KUKA KRL program: EPS_2_25618_SANMH08_A_20250918115514.src

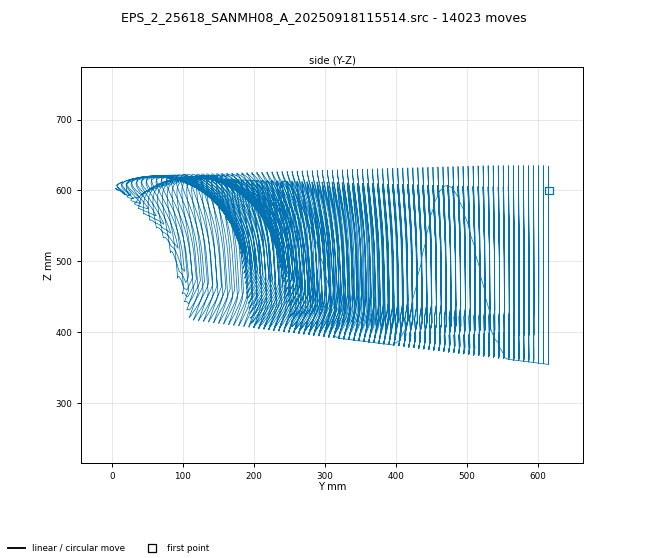
[picture p0: tool path of EPS_2_25618_SANMH08_A_20250918115514.src, 14023 of 14025 moves have a stored position in this frame; points joined in program order, loops and branches not executed]
&ACCESS RVP
&REL 4
&COMMENT QRS 19112012
&PARAM EDITMASK = *
DEF PART()
EXT BAS (BAS_COMMAND :IN,REAL :IN )
INT I
BAS (#INITMOV,0 )

;KUKA QRS Post kuka4.cps  Date:22-06-2017 !

File_ID=2843

QRS_PRE_INIT()

;Init var - Until changes are made in qrs_pre_init
Outlet_Square_prg=0
Inlet_1_Square_prg=0
Inlet_2_Square_prg=0
Inlet_3_Square_prg=0
Inlet_4_Square_prg=0
Inlet_5_Square_prg=0

Outlet_1={X 0.000, Y 530.070, Z 534.500, B 0.000, E1 0.000 }
Inlet_1={X 0.000, Y 532.210, Z 504.500, B 0.000, E1 142.000 }
Inlet_2={X 0.000, Y 532.210, Z 504.500, B 0.000, E1 248.000 }
Outlet_1_type=201
Inlet_1_type=201
Inlet_2_type=201
;QRS#1=Sidecore dimensions
;QRS#2=200-8" PVC SDR 35
;QRS#3=200-8" PVC SDR 35
;QRS#4=200-8" PVC SDR 35
;QRS#5=
;QRS#6=
;QRS#7=
;QRS#8=
;QRS#9=12-08 PSX
;QRS#10=12-08 PSX
;QRS#11=12-08 PSX
;QRS#12=
;QRS#13=
;QRS#14=
;QRS#15=
;QRS#16=1220x127x914 3'
;QRS#17=EPS Height
;QRS#18=635
;QRS#19=*
;QRS#20= UPDATED VERSION 22-06-2017
;QRS#21=*
Outlet_Square=0100
Inlet_1_Square=0100
Inlet_2_Square=0100
Inlet_3_Square=0
Inlet_4_Square=0
Inlet_5_Square=0
Mill_Square=1
Outlet_Square_Prg=204
Inlet_1_Square_prg=204
Inlet_2_Square_prg=204

QRS_INIT()

$ADVANCE=5

; T1
PTP {E1 173.609,E2 173.609}
PTP {X 0,Y 615.507,A -85,B 0,C 180,E1 173.609,E2 173.609,E3 0,E4 0,E5 0,E6 0}
QRS_SPEED_INIT()
LIN {X 0,Y 615.507,Z 600,A -85,B 0,C 180,E1 173.609,E2 173.609,E3 0,E4 0,E5 0,E6 0} C_VEL
LIN {X 0,Y 615.507,Z 364.866,A -85,B 0,C 180,E1 173.609,E2 173.609} C_VEL
LIN {X 0,Y 615.507,Z 356.684,A -85,B 0,C 180,E1 173.609,E2 173.609} C_VEL
LIN {X 0,Y 615.491,Z 354.684,A -85,B 0,C 180,E1 173.422,E2 173.422} C_VEL
LIN {X 0,Y 615.479,Z 354.687,A -85,B 0,C 180,E1 170.801,E2 170.801} C_VEL
LIN {X 0,Y 615.493,Z 354.701,A -85,B 0,C 180,E1 168.139,E2 168.139} C_VEL
LIN {X 0,Y 615.49,Z 354.683,A -85,B 0,C 180,E1 165.451,E2 165.451} C_VEL
LIN {X 0,Y 615.49,Z 354.688,A -85,B 0,C 180,E1 162.729,E2 162.729} C_VEL
LIN {X 0,Y 615.488,Z 354.691,A -85,B 0,C 180,E1 159.967,E2 159.967} C_VEL
LIN {X 0,Y 615.492,Z 354.683,A -85,B 0,C 180,E1 157.654,E2 157.654} C_VEL
LIN {X 0,Y 615.477,Z 354.689,A -85,B 0,C 180,E1 155.008,E2 155.008} C_VEL
LIN {X 0,Y 615.482,Z 354.693,A -85,B 0,C 180,E1 152.822,E2 152.822} C_VEL
LIN {X 0,Y 615.483,Z 354.693,A -85,B 0,C 180,E1 150.207,E2 150.207} C_VEL
LIN {X 0,Y 615.479,Z 354.686,A -85,B 0,C 180,E1 147.348,E2 147.348} C_VEL
LIN {X 0,Y 615.476,Z 354.783,A -85,B 0,C 180,E1 147.202,E2 147.202} C_VEL
LIN {X 0,Y 615.484,Z 371.926,A -85,B 0,C 180,E1 144.384,E2 144.384} C_VEL
LIN {X 0,Y 615.483,Z 389.625,A -85,B 0,C 180,E1 141.514,E2 141.514} C_VEL
LIN {X 0,Y 615.488,Z 393.995,A -85,B 0,C 180,E1 140.811,E2 140.811} C_VEL
LIN {X 0,Y 615.484,Z 500.165,A -85,B 0,C 180,E1 139.555,E2 139.555} C_VEL
LIN {X 0,Y 615.478,Z 513.423,A -85,B 0,C 180,E1 139.271,E2 139.271} C_VEL
LIN {X 0,Y 615.487,Z 526.153,A -85,B 0,C 180,E1 138.859,E2 138.859} C_VEL
LIN {X 0,Y 615.481,Z 537.276,A -85,B 0,C 180,E1 138.375,E2 138.375} C_VEL
LIN {X 0,Y 615.492,Z 547.938,A -85,B 0,C 180,E1 137.784,E2 137.784} C_VEL
LIN {X 0,Y 615.495,Z 558.627,A -85,B 0,C 180,E1 137.04,E2 137.04} C_VEL
LIN {X 0,Y 615.496,Z 568.483,A -85,B 0,C 180,E1 136.192,E2 136.192} C_VEL
LIN {X 0,Y 615.494,Z 577.195,A -85,B 0,C 180,E1 135.265,E2 135.265} C_VEL
LIN {X 0,Y 615.495,Z 584.222,A -85,B 0,C 180,E1 134.344,E2 134.344} C_VEL
LIN {X 0,Y 615.499,Z 590.94,A -85,B 0,C 180,E1 133.244,E2 133.244} C_VEL
LIN {X 0,Y 615.498,Z 596.401,A -85,B 0,C 180,E1 132.081,E2 132.081} C_VEL
LIN {X 0,Y 615.495,Z 599.823,A -85,B 0,C 180,E1 131.095,E2 131.095} C_VEL
LIN {X 0,Y 615.498,Z 602.292,A -85,B 0,C 180,E1 130.09,E2 130.09} C_VEL
LIN {X 0,Y 615.491,Z 603.967,A -85,B 0,C 180,E1 128.905,E2 128.905} C_VEL
LIN {X 0,Y 615.494,Z 604.381,A -85,B 0,C 180,E1 128.012,E2 128.012} C_VEL
LIN {X 0,Y 615.492,Z 603.915,A -85,B 0,C 180,E1 126.937,E2 126.937} C_VEL
LIN {X 0,Y 615.496,Z 602.323,A -85,B 0,C 180,E1 125.834,E2 125.834} C_VEL
LIN {X 0,Y 615.498,Z 599.46,A -85,B 0,C 180,E1 124.702,E2 124.702} C_VEL
LIN {X 0,Y 615.494,Z 595.146,A -85,B 0,C 180,E1 123.535,E2 123.535} C_VEL
LIN {X 0,Y 615.497,Z 589.801,A -85,B 0,C 180,E1 122.458,E2 122.458} C_VEL
LIN {X 0,Y 615.496,Z 582.973,A -85,B 0,C 180,E1 121.386,E2 121.386} C_VEL
LIN {X 0,Y 615.496,Z 574.596,A -85,B 0,C 180,E1 120.35,E2 120.35} C_VEL
LIN {X 0,Y 615.498,Z 566.188,A -85,B 0,C 180,E1 119.504,E2 119.504} C_VEL
LIN {X 0,Y 615.493,Z 555.813,A -85,B 0,C 180,E1 118.658,E2 118.658} C_VEL
LIN {X 0,Y 615.488,Z 544.388,A -85,B 0,C 180,E1 117.916,E2 117.916} C_VEL
LIN {X 0,Y 615.489,Z 532.612,A -85,B 0,C 180,E1 117.316,E2 117.316} C_VEL
LIN {X 0,Y 615.491,Z 520.703,A -85,B 0,C 180,E1 116.857,E2 116.857} C_VEL
LIN {X 0,Y 615.487,Z 508.59,A -85,B 0,C 180,E1 116.52,E2 116.52} C_VEL
LIN {X 0,Y 615.496,Z 495.123,A -85,B 0,C 180,E1 116.285,E2 116.285} C_VEL
LIN {X 0,Y 615.495,Z 393.999,A -85,B 0,C 180,E1 115.1,E2 115.1} C_VEL
LIN {X 0,Y 615.493,Z 376.959,A -85,B 0,C 180,E1 112.346,E2 112.346} C_VEL
LIN {X 0,Y 615.489,Z 359.644,A -85,B 0,C 180,E1 109.512,E2 109.512} C_VEL
LIN {X 0,Y 615.485,Z 354.686,A -85,B 0,C 180,E1 108.69,E2 108.69} C_VEL
LIN {X 0,Y 615.49,Z 354.686,A -85,B 0,C 180,E1 105.906,E2 105.906} C_VEL
LIN {X 0,Y 615.495,Z 354.694,A -85,B 0,C 180,E1 103.202,E2 103.202} C_VEL
LIN {X 0,Y 615.478,Z 354.685,A -85,B 0,C 180,E1 100.528,E2 100.528} C_VEL
LIN {X 0,Y 615.493,Z 354.69,A -85,B 0,C 180,E1 97.876,E2 97.876} C_VEL
LIN {X 0,Y 615.491,Z 354.691,A -85,B 0,C 180,E1 95.242,E2 95.242} C_VEL
LIN {X 0,Y 615.478,Z 354.685,A -85,B 0,C 180,E1 92.619,E2 92.619} C_VEL
LIN {X 0,Y 615.491,Z 354.691,A -85,B 0,C 180,E1 90.001,E2 90.001} C_VEL
LIN {X 0,Y 615.488,Z 354.692,A -85,B 0,C 180,E1 87.383,E2 87.383} C_VEL
LIN {X 0,Y 615.482,Z 354.684,A -85,B 0,C 180,E1 84.76,E2 84.76} C_VEL
LIN {X 0,Y 615.488,Z 354.692,A -85,B 0,C 180,E1 82.125,E2 82.125} C_VEL
LIN {X 0,Y 615.478,Z 354.692,A -85,B 0,C 180,E1 79.474,E2 79.474} C_VEL
LIN {X 0,Y 615.48,Z 354.685,A -85,B 0,C 180,E1 76.8,E2 76.8} C_VEL
LIN {X 0,Y 615.492,Z 354.697,A -85,B 0,C 180,E1 74.096,E2 74.096} C_VEL
LIN {X 0,Y 615.483,Z 354.686,A -85,B 0,C 180,E1 71.355,E2 71.355} C_VEL
LIN {X 0,Y 615.477,Z 354.69,A -85,B 0,C 180,E1 68.569,E2 68.569} C_VEL
LIN {X 0,Y 615.478,Z 354.692,A -85,B 0,C 180,E1 65.729,E2 65.729} C_VEL
LIN {X 0,Y 615.486,Z 354.684,A -85,B 0,C 180,E1 62.956,E2 62.956} C_VEL
LIN {X 0,Y 615.499,Z 354.699,A -85,B 0,C 180,E1 60.204,E2 60.204} C_VEL
LIN {X 0,Y 615.479,Z 354.686,A -85,B 0,C 180,E1 57.543,E2 57.543} C_VEL
LIN {X 0,Y 615.498,Z 354.68,A -85,B 0,C 180,E1 55.187,E2 55.187} C_VEL
LIN {X 0,Y 615.477,Z 354.693,A -85,B 0,C 180,E1 52.759,E2 52.759} C_VEL
LIN {X 0,Y 615.477,Z 354.69,A -85,B 0,C 180,E1 49.913,E2 49.913} C_VEL
LIN {X 0,Y 615.475,Z 354.686,A -85,B 0,C 180,E1 47.648,E2 47.648} C_VEL
LIN {X 0,Y 615.488,Z 354.69,A -85,B 0,C 180,E1 44.933,E2 44.933} C_VEL
LIN {X 0,Y 615.486,Z 354.688,A -85,B 0,C 180,E1 42.082,E2 42.082} C_VEL
LIN {X 0,Y 615.492,Z 354.846,A -85,B 0,C 180,E1 41.191,E2 41.191} C_VEL
LIN {X 0,Y 615.494,Z 371.303,A -85,B 0,C 180,E1 38.485,E2 38.485} C_VEL
LIN {X 0,Y 615.498,Z 388.993,A -85,B 0,C 180,E1 35.615,E2 35.615} C_VEL
LIN {X 0,Y 615.487,Z 393.968,A -85,B 0,C 180,E1 34.815,E2 34.815} C_VEL
LIN {X 0,Y 615.488,Z 501.254,A -85,B 0,C 180,E1 33.537,E2 33.537} C_VEL
LIN {X 0,Y 615.491,Z 514.682,A -85,B 0,C 180,E1 33.236,E2 33.236} C_VEL
LIN {X 0,Y 615.488,Z 526.503,A -85,B 0,C 180,E1 32.846,E2 32.846} C_VEL
LIN {X 0,Y 615.495,Z 538.108,A -85,B 0,C 180,E1 32.334,E2 32.334} C_VEL
LIN {X 0,Y 615.481,Z 549.464,A -85,B 0,C 180,E1 31.686,E2 31.686} C_VEL
LIN {X 0,Y 615.498,Z 560.16,A -85,B 0,C 180,E1 30.919,E2 30.919} C_VEL
LIN {X 0,Y 615.499,Z 568.823,A -85,B 0,C 180,E1 30.16,E2 30.16} C_VEL
LIN {X 0,Y 615.497,Z 577.573,A -85,B 0,C 180,E1 29.218,E2 29.218} C_VEL
LIN {X 0,Y 615.497,Z 585.301,A -85,B 0,C 180,E1 28.184,E2 28.184} C_VEL
LIN {X 0,Y 615.494,Z 591.99,A -85,B 0,C 180,E1 27.049,E2 27.049} C_VEL
LIN {X 0,Y 615.498,Z 596.407,A -85,B 0,C 180,E1 26.079,E2 26.079} C_VEL
LIN {X 0,Y 615.493,Z 600.114,A -85,B 0,C 180,E1 24.992,E2 24.992} C_VEL
LIN {X 0,Y 615.495,Z 602.448,A -85,B 0,C 180,E1 24.013,E2 24.013} C_VEL
LIN {X 0,Y 615.495,Z 604.008,A -85,B 0,C 180,E1 22.844,E2 22.844} C_VEL
LIN {X 0,Y 615.496,Z 604.351,A -85,B 0,C 180,E1 22.136,E2 22.136} C_VEL
LIN {X 0,Y 615.497,Z 604.263,A -85,B 0,C 180,E1 21.432,E2 21.432} C_VEL
LIN {X 0,Y 615.496,Z 603.481,A -85,B 0,C 180,E1 20.563,E2 20.563} C_VEL
LIN {X 0,Y 615.495,Z 601.235,A -85,B 0,C 180,E1 19.338,E2 19.338} C_VEL
LIN {X 0,Y 615.499,Z 598.102,A -85,B 0,C 180,E1 18.284,E2 18.284} C_VEL
LIN {X 0,Y 615.496,Z 593.986,A -85,B 0,C 180,E1 17.27,E2 17.27} C_VEL
LIN {X 0,Y 615.497,Z 588.127,A -85,B 0,C 180,E1 16.172,E2 16.172} C_VEL
LIN {X 0,Y 615.496,Z 580.518,A -85,B 0,C 180,E1 15.056,E2 15.056} C_VEL
LIN {X 0,Y 615.498,Z 572.231,A -85,B 0,C 180,E1 14.094,E2 14.094} C_VEL
LIN {X 0,Y 615.499,Z 562.722,A -85,B 0,C 180,E1 13.201,E2 13.201} C_VEL
LIN {X 0,Y 615.491,Z 552.852,A -85,B 0,C 180,E1 12.446,E2 12.446} C_VEL
LIN {X 0,Y 615.475,Z 541.927,A -85,B 0,C 180,E1 11.778,E2 11.778} C_VEL
LIN {X 0,Y 615.497,Z 529.711,A -85,B 0,C 180,E1 11.193,E2 11.193} C_VEL
LIN {X 0,Y 615.486,Z 517.603,A -85,B 0,C 180,E1 10.757,E2 10.757} C_VEL
LIN {X 0,Y 615.499,Z 505.077,A -85,B 0,C 180,E1 10.444,E2 10.444} C_VEL
LIN {X 0,Y 615.493,Z 489.201,A -85,B 0,C 180,E1 10.215,E2 10.215} C_VEL
LIN {X 0,Y 615.491,Z 393.971,A -85,B 0,C 180,E1 9.095,E2 9.095} C_VEL
LIN {X 0,Y 615.493,Z 376.229,A -85,B 0,C 180,E1 6.228,E2 6.228} C_VEL
LIN {X 0,Y 615.49,Z 360.181,A -85,B 0,C 180,E1 3.601,E2 3.601} C_VEL
LIN {X 0,Y 615.49,Z 354.685,A -85,B 0,C 180,E1 2.659,E2 2.659} C_VEL
LIN {X 0,Y 615.477,Z 354.688,A -85,B 0,C 180,E1 0,E2 0} C_VEL
LIN {X 0,Y 615.493,Z 354.698,A -85,B 0,C 180,E1 -2.618,E2 -2.618} C_VEL
LIN {X 0,Y 615.484,Z 354.685,A -85,B 0,C 180,E1 -5.241,E2 -5.241} C_VEL
LIN {X 0,Y 615.482,Z 354.69,A -85,B 0,C 180,E1 -7.876,E2 -7.876} C_VEL
LIN {X 0,Y 615.493,Z 354.693,A -85,B 0,C 180,E1 -10.527,E2 -10.527} C_VEL
LIN {X 0,Y 615.484,Z 354.684,A -85,B 0,C 180,E1 -13.201,E2 -13.201} C_VEL
LIN {X 0,Y 615.49,Z 354.695,A -85,B 0,C 180,E1 -15.905,E2 -15.905} C_VEL
LIN {X 0,Y 615.483,Z 354.687,A -85,B 0,C 180,E1 -18.646,E2 -18.646} C_VEL
LIN {X 0,Y 615.496,Z 354.686,A -85,B 0,C 180,E1 -21.432,E2 -21.432} C_VEL
LIN {X 0,Y 615.494,Z 354.689,A -85,B 0,C 180,E1 -24.272,E2 -24.272} C_VEL
LIN {X 0,Y 615.477,Z 354.687,A -85,B 0,C 180,E1 -27.046,E2 -27.046} C_VEL
LIN {X 0,Y 615.495,Z 354.698,A -85,B 0,C 180,E1 -29.798,E2 -29.798} C_VEL
LIN {X 0,Y 615.489,Z 354.683,A -85,B 0,C 180,E1 -32.457,E2 -32.457} C_VEL
LIN {X 0,Y 615.477,Z 354.687,A -85,B 0,C 180,E1 -34.816,E2 -34.816} C_VEL
LIN {X 0,Y 615.488,Z 354.695,A -85,B 0,C 180,E1 -37.242,E2 -37.242} C_VEL
LIN {X 0,Y 615.486,Z 354.685,A -85,B 0,C 180,E1 -40.091,E2 -40.091} C_VEL
LIN {X 0,Y 615.493,Z 354.682,A -85,B 0,C 180,E1 -42.353,E2 -42.353} C_VEL
LIN {X 0,Y 615.48,Z 354.699,A -85,B 0,C 180,E1 -45.069,E2 -45.069} C_VEL
LIN {X 0,Y 615.48,Z 354.686,A -85,B 0,C 180,E1 -47.921,E2 -47.921} C_VEL
LIN {X 0,Y 615.494,Z 354.682,A -85,B 0,C 180,E1 -50.252,E2 -50.252} C_VEL
LIN {X 0,Y 615.492,Z 354.699,A -85,B 0,C 180,E1 -53.063,E2 -53.063} C_VEL
LIN {X 0,Y 615.491,Z 354.69,A -85,B 0,C 180,E1 -55.299,E2 -55.299} C_VEL
LIN {X 0,Y 615.477,Z 354.686,A -85,B 0,C 180,E1 -57.671,E2 -57.671} C_VEL
LIN {X 0,Y 615.498,Z 354.684,A -85,B 0,C 180,E1 -60.204,E2 -60.204} C_VEL
LIN {X 0,Y 615.493,Z 354.693,A -85,B 0,C 180,E1 -62.954,E2 -62.954} C_VEL
LIN {X 0,Y 615.478,Z 354.685,A -85,B 0,C 180,E1 -65.729,E2 -65.729} C_VEL
LIN {X 0,Y 615.481,Z 354.768,A -85,B 0,C 180,E1 -67.839,E2 -67.839} C_VEL
LIN {X 0,Y 615.478,Z 373.827,A -85,B 0,C 180,E1 -70.489,E2 -70.489} C_VEL
LIN {X 0,Y 615.488,Z 393.936,A -85,B 0,C 180,E1 -73.244,E2 -73.244} C_VEL
LIN {X 0,Y 615.494,Z 415.278,A -85,B 0,C 180,E1 -76.127,E2 -76.127} C_VEL
LIN {X 0,Y 615.497,Z 422.647,A -85,B 0,C 180,E1 -77.115,E2 -77.115} C_VEL
LIN {X 0,Y 615.479,Z 530.885,A -85,B 0,C 180,E1 -78.411,E2 -78.411} C_VEL
LIN {X 0,Y 615.478,Z 543.381,A -85,B 0,C 180,E1 -78.683,E2 -78.683} C_VEL
LIN {X 0,Y 615.491,Z 556.57,A -85,B 0,C 180,E1 -79.111,E2 -79.111} C_VEL
LIN {X 0,Y 615.478,Z 568.497,A -85,B 0,C 180,E1 -79.64,E2 -79.64} C_VEL
LIN {X 0,Y 615.487,Z 580.01,A -85,B 0,C 180,E1 -80.305,E2 -80.305} C_VEL
LIN {X 0,Y 615.499,Z 590.353,A -85,B 0,C 180,E1 -81.051,E2 -81.051} C_VEL
LIN {X 0,Y 615.497,Z 598.822,A -85,B 0,C 180,E1 -81.795,E2 -81.795} C_VEL
LIN {X 0,Y 615.497,Z 607.973,A -85,B 0,C 180,E1 -82.785,E2 -82.785} C_VEL
LIN {X 0,Y 615.497,Z 615.321,A -85,B 0,C 180,E1 -83.774,E2 -83.774} C_VEL
LIN {X 0,Y 615.499,Z 621.209,A -85,B 0,C 180,E1 -84.76,E2 -84.76} C_VEL
LIN {X 0,Y 615.493,Z 625.855,A -85,B 0,C 180,E1 -85.744,E2 -85.744} C_VEL
LIN {X 0,Y 615.495,Z 629.401,A -85,B 0,C 180,E1 -86.728,E2 -86.728} C_VEL
LIN {X 0,Y 615.497,Z 631.235,A -85,B 0,C 180,E1 -87.383,E2 -87.383} C_VEL
LIN {X 0,Y 615.497,Z 632.609,A -85,B 0,C 180,E1 -88.038,E2 -88.038} C_VEL
LIN {X 0,Y 615.496,Z 634.174,A -85,B 0,C 180,E1 -89.347,E2 -89.347} C_VEL
LIN {X 0,Y 615.494,Z 634.389,A -85,B 0,C 180,E1 -90.001,E2 -90.001} C_VEL
LIN {X 0,Y 615.496,Z 633.579,A -85,B 0,C 180,E1 -91.309,E2 -91.309} C_VEL
LIN {X 0,Y 615.498,Z 632.607,A -85,B 0,C 180,E1 -91.964,E2 -91.964} C_VEL
LIN {X 0,Y 615.497,Z 631.231,A -85,B 0,C 180,E1 -92.619,E2 -92.619} C_VEL
LIN {X 0,Y 615.496,Z 628.347,A -85,B 0,C 180,E1 -93.601,E2 -93.601} C_VEL
LIN {X 0,Y 615.498,Z 624.438,A -85,B 0,C 180,E1 -94.585,E2 -94.585} C_VEL
LIN {X 0,Y 615.499,Z 619.4,A -85,B 0,C 180,E1 -95.57,E2 -95.57} C_VEL
LIN {X 0,Y 615.497,Z 612.869,A -85,B 0,C 180,E1 -96.583,E2 -96.583} C_VEL
LIN {X 0,Y 615.497,Z 605.126,A -85,B 0,C 180,E1 -97.546,E2 -97.546} C_VEL
LIN {X 0,Y 615.498,Z 597.036,A -85,B 0,C 180,E1 -98.372,E2 -98.372} C_VEL
LIN {X 0,Y 615.499,Z 587.157,A -85,B 0,C 180,E1 -99.199,E2 -99.199} C_VEL
LIN {X 0,Y 615.488,Z 575.968,A -85,B 0,C 180,E1 -99.946,E2 -99.946} C_VEL
LIN {X 0,Y 615.481,Z 565.007,A -85,B 0,C 180,E1 -100.528,E2 -100.528} C_VEL
LIN {X 0,Y 615.49,Z 552.438,A -85,B 0,C 180,E1 -101.042,E2 -101.042} C_VEL
LIN {X 0,Y 615.477,Z 540.034,A -85,B 0,C 180,E1 -101.403,E2 -101.403} C_VEL
LIN {X 0,Y 615.481,Z 526.412,A -85,B 0,C 180,E1 -101.653,E2 -101.653} C_VEL
LIN {X 0,Y 615.497,Z 422.634,A -85,B 0,C 180,E1 -102.887,E2 -102.887} C_VEL
LIN {X 0,Y 615.486,Z 401.46,A -85,B 0,C 180,E1 -105.736,E2 -105.736} C_VEL
LIN {X 0,Y 615.478,Z 381.601,A -85,B 0,C 180,E1 -108.441,E2 -108.441} C_VEL
LIN {X 0,Y 615.492,Z 361.234,A -85,B 0,C 180,E1 -111.257,E2 -111.257} C_VEL
LIN {X 0,Y 615.48,Z 354.686,A -85,B 0,C 180,E1 -112.189,E2 -112.189} C_VEL
LIN {X 0,Y 615.494,Z 354.688,A -85,B 0,C 180,E1 -114.992,E2 -114.992} C_VEL
LIN {X 0,Y 615.487,Z 354.687,A -85,B 0,C 180,E1 -117.916,E2 -117.916} C_VEL
LIN {X 0,Y 615.476,Z 354.686,A -85,B 0,C 180,E1 -120.161,E2 -120.161} C_VEL
LIN {X 0,Y 615.479,Z 354.685,A -85,B 0,C 180,E1 -122.459,E2 -122.459} C_VEL
LIN {X 0,Y 615.499,Z 354.687,A -85,B 0,C 180,E1 -124.815,E2 -124.815} C_VEL
LIN {X 0,Y 615.496,Z 354.698,A -85,B 0,C 180,E1 -127.242,E2 -127.242} C_VEL
LIN {X 0,Y 615.476,Z 354.685,A -85,B 0,C 180,E1 -130.087,E2 -130.087} C_VEL
LIN {X 0,Y 615.476,Z 354.687,A -85,B 0,C 180,E1 -132.355,E2 -132.355} C_VEL
LIN {X 0,Y 615.493,Z 354.699,A -85,B 0,C 180,E1 -135.069,E2 -135.069} C_VEL
LIN {X 0,Y 615.486,Z 354.683,A -85,B 0,C 180,E1 -137.921,E2 -137.921} C_VEL
LIN {X 0,Y 615.477,Z 354.688,A -85,B 0,C 180,E1 -140.249,E2 -140.249} C_VEL
LIN {X 0,Y 615.478,Z 354.697,A -85,B 0,C 180,E1 -143.065,E2 -143.065} C_VEL
LIN {X 0,Y 615.481,Z 354.685,A -85,B 0,C 180,E1 -145.978,E2 -145.978} C_VEL
LIN {X 0,Y 615.476,Z 354.692,A -85,B 0,C 180,E1 -148.314,E2 -148.314} C_VEL
LIN {X 0,Y 615.486,Z 354.7,A -85,B 0,C 180,E1 -150.594,E2 -150.594} C_VEL
LIN {X 0,Y 615.492,Z 354.682,A -85,B 0,C 180,E1 -153.556,E2 -153.556} C_VEL
LIN {X 0,Y 615.487,Z 354.699,A -85,B 0,C 180,E1 -156.444,E2 -156.444} C_VEL
LIN {X 0,Y 615.477,Z 354.686,A -85,B 0,C 180,E1 -159.269,E2 -159.269} C_VEL
LIN {X 0,Y 615.482,Z 354.691,A -85,B 0,C 180,E1 -162.043,E2 -162.043} C_VEL
LIN {X 0,Y 615.486,Z 354.691,A -85,B 0,C 180,E1 -164.774,E2 -164.774} C_VEL
LIN {X 0,Y 615.486,Z 354.683,A -85,B 0,C 180,E1 -167.47,E2 -167.47} C_VEL
LIN {X 0,Y 615.493,Z 354.697,A -85,B 0,C 180,E1 -170.138,E2 -170.138} C_VEL
LIN {X 0,Y 615.483,Z 354.687,A -85,B 0,C 180,E1 -172.784,E2 -172.784} C_VEL
LIN {X 0,Y 615.491,Z 354.683,A -85,B 0,C 180,E1 -175.416,E2 -175.416} C_VEL
LIN {X 0,Y 615.497,Z 354.698,A -85,B 0,C 180,E1 -178.037,E2 -178.037} C_VEL
LIN {X 0,Y 615.483,Z 354.687,A -85,B 0,C 180,E1 -180.654,E2 -180.654} C_VEL
LIN {X 0,Y 615.485,Z 354.685,A -85,B 0,C 180,E1 -183.273,E2 -183.273} C_VEL
LIN {X 0,Y 615.497,Z 354.699,A -85,B 0,C 180,E1 -185.899,E2 -185.899} C_VEL
LIN {X 0,Y 615.491,Z 354.684,A -85,B 0,C 180,E1 -186.578,E2 -186.578} C_VEL
LIN {X 0,Y 614.809,Z 354.833,A -85,B 0,C 180,E1 -187.124,E2 -187.124} C_VEL
LIN {X 0,Y 611.966,Z 355.259,A -85,B 0,C 180,E1 -188.009,E2 -188.009} C_VEL
LIN {X 0,Y 609.575,Z 355.564,A -85,B 0,C 180,E1 -188.722,E2 -188.722} C_VEL
LIN {X 0,Y 608.546,Z 355.679,A -85,B 0,C 180,E1 -189.272,E2 -189.272} C_VEL
LIN {X 0,Y 608.46,Z 355.689,A -85,B 0,C 180,E1 -189.458,E2 -189.458} C_VEL
LIN {X 0,Y 608.467,Z 355.693,A -85,B 0,C 180,E1 -192,E2 -192} C_VEL
LIN {X 0,Y 608.478,Z 355.684,A -85,B 0,C 180,E1 -194.721,E2 -194.721} C_VEL
LIN {X 0,Y 608.455,Z 355.694,A -85,B 0,C 180,E1 -197.477,E2 -197.477} C_VEL
LIN {X 0,Y 608.464,Z 355.688,A -85,B 0,C 180,E1 -200.274,E2 -200.274} C_VEL
LIN {X 0,Y 608.464,Z 355.686,A -85,B 0,C 180,E1 -202.476,E2 -202.476} C_VEL
LIN {X 0,Y 608.453,Z 355.687,A -85,B 0,C 180,E1 -204.571,E2 -204.571} C_VEL
LIN {X 0,Y 608.476,Z 355.69,A -85,B 0,C 180,E1 -207.206,E2 -207.206} C_VEL
LIN {X 0,Y 608.467,Z 355.688,A -85,B 0,C 180,E1 -209.971,E2 -209.971} C_VEL
LIN {X 0,Y 608.469,Z 355.747,A -85,B 0,C 180,E1 -212.721,E2 -212.721} C_VEL
LIN {X 0,Y 608.479,Z 372.306,A -85,B 0,C 180,E1 -215.468,E2 -215.468} C_VEL
LIN {X 0,Y 608.474,Z 389.259,A -85,B 0,C 180,E1 -218.24,E2 -218.24} C_VEL
LIN {X 0,Y 608.468,Z 394.334,A -85,B 0,C 180,E1 -219.043,E2 -219.043} C_VEL
LIN {X 0,Y 608.56,Z 500.806,A -85,B 0,C 180,E1 -220.319,E2 -220.319} C_VEL
LIN {X 0,Y 608.524,Z 513.981,A -85,B 0,C 180,E1 -220.61,E2 -220.61} C_VEL
LIN {X 0,Y 608.508,Z 526.119,A -85,B 0,C 180,E1 -221.008,E2 -221.008} C_VEL
LIN {X 0,Y 608.515,Z 537.812,A -85,B 0,C 180,E1 -221.523,E2 -221.523} C_VEL
LIN {X 0,Y 608.496,Z 549.609,A -85,B 0,C 180,E1 -222.198,E2 -222.198} C_VEL
LIN {X 0,Y 608.469,Z 560.192,A -85,B 0,C 180,E1 -222.959,E2 -222.959} C_VEL
LIN {X 0,Y 608.477,Z 568.796,A -85,B 0,C 180,E1 -223.714,E2 -223.714} C_VEL
LIN {X 0,Y 608.46,Z 577.541,A -85,B 0,C 180,E1 -224.648,E2 -224.648} C_VEL
LIN {X 0,Y 608.45,Z 585.685,A -85,B 0,C 180,E1 -225.737,E2 -225.737} C_VEL
LIN {X 0,Y 608.437,Z 591.419,A -85,B 0,C 180,E1 -226.695,E2 -226.695} C_VEL
LIN {X 0,Y 608.437,Z 596.069,A -85,B 0,C 180,E1 -227.669,E2 -227.669} C_VEL
LIN {X 0,Y 608.432,Z 600.233,A -85,B 0,C 180,E1 -228.821,E2 -228.821} C_VEL
LIN {X 0,Y 608.422,Z 602.465,A -85,B 0,C 180,E1 -229.694,E2 -229.694} C_VEL
LIN {X 0,Y 608.423,Z 604.169,A -85,B 0,C 180,E1 -230.708,E2 -230.708} C_VEL
LIN {X 0,Y 608.414,Z 604.941,A -85,B 0,C 180,E1 -231.767,E2 -231.767} C_VEL
LIN {X 0,Y 608.43,Z 604.514,A -85,B 0,C 180,E1 -233.083,E2 -233.083} C_VEL
LIN {X 0,Y 608.426,Z 603.323,A -85,B 0,C 180,E1 -233.958,E2 -233.958} C_VEL
LIN {X 0,Y 608.426,Z 600.729,A -85,B 0,C 180,E1 -235.098,E2 -235.098} C_VEL
LIN {X 0,Y 608.435,Z 596.474,A -85,B 0,C 180,E1 -236.327,E2 -236.327} C_VEL
LIN {X 0,Y 608.435,Z 590.944,A -85,B 0,C 180,E1 -237.482,E2 -237.482} C_VEL
LIN {X 0,Y 608.44,Z 584.781,A -85,B 0,C 180,E1 -238.487,E2 -238.487} C_VEL
LIN {X 0,Y 608.457,Z 577.442,A -85,B 0,C 180,E1 -239.454,E2 -239.454} C_VEL
LIN {X 0,Y 608.462,Z 568.439,A -85,B 0,C 180,E1 -240.41,E2 -240.41} C_VEL
LIN {X 0,Y 608.497,Z 559.112,A -85,B 0,C 180,E1 -241.216,E2 -241.216} C_VEL
LIN {X 0,Y 608.501,Z 549.146,A -85,B 0,C 180,E1 -241.923,E2 -241.923} C_VEL
LIN {X 0,Y 608.511,Z 537.534,A -85,B 0,C 180,E1 -242.581,E2 -242.581} C_VEL
LIN {X 0,Y 608.514,Z 525.264,A -85,B 0,C 180,E1 -243.114,E2 -243.114} C_VEL
LIN {X 0,Y 608.54,Z 512.165,A -85,B 0,C 180,E1 -243.53,E2 -243.53} C_VEL
LIN {X 0,Y 608.567,Z 499.905,A -85,B 0,C 180,E1 -243.785,E2 -243.785} C_VEL
LIN {X 0,Y 608.513,Z 394.562,A -85,B 0,C 180,E1 -245.044,E2 -245.044} C_VEL
LIN {X 0,Y 608.482,Z 394.094,A -85,B 0,C 180,E1 -245.065,E2 -245.065} C_VEL
LIN {X 0,Y 608.494,Z 376.377,A -85,B 0,C 180,E1 -247.952,E2 -247.952} C_VEL
LIN {X 0,Y 608.506,Z 359.26,A -85,B 0,C 180,E1 -250.781,E2 -250.781} C_VEL
LIN {X 0,Y 608.478,Z 355.686,A -85,B 0,C 180,E1 -251.383,E2 -251.383} C_VEL
LIN {X 0,Y 608.46,Z 355.687,A -85,B 0,C 180,E1 -253.905,E2 -253.905} C_VEL
LIN {X 0,Y 608.472,Z 355.695,A -85,B 0,C 180,E1 -256.643,E2 -256.643} C_VEL
LIN {X 0,Y 608.461,Z 355.687,A -85,B 0,C 180,E1 -259.349,E2 -259.349} C_VEL
LIN {X 0,Y 608.483,Z 355.687,A -85,B 0,C 180,E1 -262.032,E2 -262.032} C_VEL
LIN {X 0,Y 608.471,Z 355.691,A -85,B 0,C 180,E1 -264.697,E2 -264.697} C_VEL
LIN {X 0,Y 608.471,Z 355.685,A -85,B 0,C 180,E1 -267.351,E2 -267.351} C_VEL
LIN {X 0,Y 608.482,Z 355.689,A -85,B 0,C 180,E1 -269.999,E2 -269.999} C_VEL
LIN {X 0,Y 608.479,Z 355.689,A -85,B 0,C 180,E1 -272.647,E2 -272.647} C_VEL
LIN {X 0,Y 608.463,Z 355.686,A -85,B 0,C 180,E1 -275.301,E2 -275.301} C_VEL
LIN {X 0,Y 608.479,Z 355.691,A -85,B 0,C 180,E1 -277.966,E2 -277.966} C_VEL
LIN {X 0,Y 608.468,Z 355.686,A -85,B 0,C 180,E1 -280.953,E2 -280.953} C_VEL
LIN {X 0,Y 608.461,Z 355.687,A -85,B 0,C 180,E1 -283.355,E2 -283.355} C_VEL
LIN {X 0,Y 608.461,Z 355.696,A -85,B 0,C 180,E1 -286.093,E2 -286.093} C_VEL
LIN {X 0,Y 608.453,Z 355.687,A -85,B 0,C 180,E1 -288.869,E2 -288.869} C_VEL
LIN {X 0,Y 608.462,Z 355.693,A -85,B 0,C 180,E1 -291.691,E2 -291.691} C_VEL
LIN {X 0,Y 608.45,Z 355.689,A -85,B 0,C 180,E1 -294.57,E2 -294.57} C_VEL
LIN {X 0,Y 608.475,Z 355.686,A -85,B 0,C 180,E1 -297.206,E2 -297.206} C_VEL
LIN {X 0,Y 608.471,Z 355.692,A -85,B 0,C 180,E1 -299.971,E2 -299.971} C_VEL
LIN {X 0,Y 608.455,Z 355.688,A -85,B 0,C 180,E1 -302.521,E2 -302.521} C_VEL
LIN {X 0,Y 608.453,Z 355.692,A -85,B 0,C 180,E1 -305.276,E2 -305.276} C_VEL
LIN {X 0,Y 608.464,Z 355.687,A -85,B 0,C 180,E1 -308.239,E2 -308.239} C_VEL
LIN {X 0,Y 608.445,Z 355.689,A -85,B 0,C 180,E1 -310.328,E2 -310.328} C_VEL
LIN {X 0,Y 608.476,Z 355.692,A -85,B 0,C 180,E1 -313.309,E2 -313.309} C_VEL
LIN {X 0,Y 608.468,Z 355.687,A -85,B 0,C 180,E1 -316.13,E2 -316.13} C_VEL
LIN {X 0,Y 608.497,Z 355.702,A -85,B 0,C 180,E1 -318.715,E2 -318.715} C_VEL
LIN {X 0,Y 608.487,Z 371.969,A -85,B 0,C 180,E1 -321.413,E2 -321.413} C_VEL
LIN {X 0,Y 608.479,Z 389.856,A -85,B 0,C 180,E1 -324.338,E2 -324.338} C_VEL
LIN {X 0,Y 608.46,Z 394.135,A -85,B 0,C 180,E1 -325.031,E2 -325.031} C_VEL
LIN {X 0,Y 608.535,Z 501.608,A -85,B 0,C 180,E1 -326.333,E2 -326.333} C_VEL
LIN {X 0,Y 608.55,Z 515.205,A -85,B 0,C 180,E1 -326.644,E2 -326.644} C_VEL
LIN {X 0,Y 608.509,Z 527.86,A -85,B 0,C 180,E1 -327.074,E2 -327.074} C_VEL
LIN {X 0,Y 608.508,Z 538.903,A -85,B 0,C 180,E1 -327.579,E2 -327.579} C_VEL
LIN {X 0,Y 608.482,Z 549.629,A -85,B 0,C 180,E1 -328.199,E2 -328.199} C_VEL
LIN {X 0,Y 608.489,Z 560.505,A -85,B 0,C 180,E1 -328.984,E2 -328.984} C_VEL
LIN {X 0,Y 608.486,Z 569.436,A -85,B 0,C 180,E1 -329.774,E2 -329.774} C_VEL
LIN {X 0,Y 608.46,Z 577.142,A -85,B 0,C 180,E1 -330.6,E2 -330.6} C_VEL
LIN {X 0,Y 608.447,Z 584.468,A -85,B 0,C 180,E1 -331.557,E2 -331.557} C_VEL
LIN {X 0,Y 608.438,Z 590.253,A -85,B 0,C 180,E1 -332.481,E2 -332.481} C_VEL
LIN {X 0,Y 608.455,Z 595.758,A -85,B 0,C 180,E1 -333.596,E2 -333.596} C_VEL
LIN {X 0,Y 608.437,Z 599.842,A -85,B 0,C 180,E1 -334.698,E2 -334.698} C_VEL
LIN {X 0,Y 608.424,Z 602.816,A -85,B 0,C 180,E1 -335.856,E2 -335.856} C_VEL
LIN {X 0,Y 608.431,Z 604.365,A -85,B 0,C 180,E1 -336.875,E2 -336.875} C_VEL
LIN {X 0,Y 608.423,Z 604.9,A -85,B 0,C 180,E1 -337.592,E2 -337.592} C_VEL
LIN {X 0,Y 608.416,Z 604.945,A -85,B 0,C 180,E1 -338.306,E2 -338.306} C_VEL
LIN {X 0,Y 608.438,Z 604.236,A -85,B 0,C 180,E1 -339.325,E2 -339.325} C_VEL
LIN {X 0,Y 608.416,Z 602.398,A -85,B 0,C 180,E1 -340.428,E2 -340.428} C_VEL
LIN {X 0,Y 608.425,Z 600.158,A -85,B 0,C 180,E1 -341.293,E2 -341.293} C_VEL
LIN {X 0,Y 608.428,Z 595.637,A -85,B 0,C 180,E1 -342.523,E2 -342.523} C_VEL
LIN {X 0,Y 608.437,Z 589.798,A -85,B 0,C 180,E1 -343.691,E2 -343.691} C_VEL
LIN {X 0,Y 608.456,Z 582.824,A -85,B 0,C 180,E1 -344.765,E2 -344.765} C_VEL
LIN {X 0,Y 608.458,Z 574.468,A -85,B 0,C 180,E1 -345.792,E2 -345.792} C_VEL
LIN {X 0,Y 608.481,Z 565.945,A -85,B 0,C 180,E1 -346.644,E2 -346.644} C_VEL
LIN {X 0,Y 608.49,Z 555.441,A -85,B 0,C 180,E1 -347.493,E2 -347.493} C_VEL
LIN {X 0,Y 608.471,Z 545.104,A -85,B 0,C 180,E1 -348.169,E2 -348.169} C_VEL
LIN {X 0,Y 608.531,Z 534.17,A -85,B 0,C 180,E1 -348.742,E2 -348.742} C_VEL
LIN {X 0,Y 608.537,Z 523.099,A -85,B 0,C 180,E1 -349.195,E2 -349.195} C_VEL
LIN {X 0,Y 608.531,Z 510.906,A -85,B 0,C 180,E1 -349.562,E2 -349.562} C_VEL
LIN {X 0,Y 608.553,Z 497.848,A -85,B 0,C 180,E1 -349.814,E2 -349.814} C_VEL
LIN {X 0,Y 608.459,Z 394.19,A -85,B 0,C 180,E1 -351.05,E2 -351.05} C_VEL
LIN {X 0,Y 608.491,Z 377.157,A -85,B 0,C 180,E1 -353.824,E2 -353.824} C_VEL
LIN {X 0,Y 608.512,Z 359.81,A -85,B 0,C 180,E1 -356.689,E2 -356.689} C_VEL
LIN {X 0,Y 608.462,Z 355.688,A -85,B 0,C 180,E1 -357.393,E2 -357.393} C_VEL
LIN {X 0,Y 608.468,Z 355.688,A -85,B 0,C 180,E1 -360,E2 -360} C_VEL
LIN {X 0,Y 608.482,Z 355.692,A -85,B 0,C 180,E1 -362.648,E2 -362.648} C_VEL
LIN {X 0,Y 608.462,Z 355.687,A -85,B 0,C 180,E1 -365.302,E2 -365.302} C_VEL
LIN {X 0,Y 608.473,Z 355.689,A -85,B 0,C 180,E1 -367.967,E2 -367.967} C_VEL
LIN {X 0,Y 608.465,Z 355.69,A -85,B 0,C 180,E1 -370.65,E2 -370.65} C_VEL
LIN {X 0,Y 608.462,Z 355.687,A -85,B 0,C 180,E1 -373.356,E2 -373.356} C_VEL
LIN {X 0,Y 608.485,Z 355.694,A -85,B 0,C 180,E1 -376.093,E2 -376.093} C_VEL
LIN {X 0,Y 608.451,Z 355.688,A -85,B 0,C 180,E1 -378.87,E2 -378.87} C_VEL
LIN {X 0,Y 608.477,Z 355.691,A -85,B 0,C 180,E1 -381.691,E2 -381.691} C_VEL
LIN {X 0,Y 608.452,Z 355.689,A -85,B 0,C 180,E1 -384.571,E2 -384.571} C_VEL
LIN {X 0,Y 608.473,Z 355.687,A -85,B 0,C 180,E1 -387.209,E2 -387.209} C_VEL
LIN {X 0,Y 608.472,Z 355.691,A -85,B 0,C 180,E1 -389.975,E2 -389.975} C_VEL
LIN {X 0,Y 608.459,Z 355.688,A -85,B 0,C 180,E1 -392.88,E2 -392.88} C_VEL
LIN {X 0,Y 608.439,Z 355.695,A -85,B 0,C 180,E1 -395.278,E2 -395.278} C_VEL
LIN {X 0,Y 608.467,Z 355.691,A -85,B 0,C 180,E1 -397.747,E2 -397.747} C_VEL
LIN {X 0,Y 608.449,Z 355.688,A -85,B 0,C 180,E1 -400.331,E2 -400.331} C_VEL
LIN {X 0,Y 608.483,Z 355.694,A -85,B 0,C 180,E1 -403.312,E2 -403.312} C_VEL
LIN {X 0,Y 608.467,Z 355.686,A -85,B 0,C 180,E1 -406.132,E2 -406.132} C_VEL
LIN {X 0,Y 608.449,Z 355.693,A -85,B 0,C 180,E1 -408.825,E2 -408.825} C_VEL
LIN {X 0,Y 608.473,Z 355.689,A -85,B 0,C 180,E1 -411.414,E2 -411.414} C_VEL
LIN {X 0,Y 608.475,Z 355.685,A -85,B 0,C 180,E1 -413.951,E2 -413.951} C_VEL
LIN {X 0,Y 608.465,Z 355.688,A -85,B 0,C 180,E1 -416.331,E2 -416.331} C_VEL
LIN {X 0,Y 608.478,Z 355.693,A -85,B 0,C 180,E1 -418.728,E2 -418.728} C_VEL
LIN {X 0,Y 608.469,Z 355.687,A -85,B 0,C 180,E1 -421.381,E2 -421.381} C_VEL
LIN {X 0,Y 608.447,Z 355.689,A -85,B 0,C 180,E1 -423.966,E2 -423.966} C_VEL
LIN {X 0,Y 608.468,Z 355.689,A -85,B 0,C 180,E1 -426.156,E2 -426.156} C_VEL
LIN {X 0,Y 608.468,Z 355.741,A -85,B 0,C 180,E1 -427.707,E2 -427.707} C_VEL
LIN {X 0,Y 608.541,Z 371.325,A -85,B 0,C 180,E1 -429.906,E2 -429.906} C_VEL
LIN {X 0,Y 608.527,Z 391.474,A -85,B 0,C 180,E1 -432.7,E2 -432.7} C_VEL
LIN {X 0,Y 608.494,Z 412.883,A -85,B 0,C 180,E1 -435.623,E2 -435.623} C_VEL
LIN {X 0,Y 608.477,Z 422.8,A -85,B 0,C 180,E1 -436.963,E2 -436.963} C_VEL
LIN {X 0,Y 608.569,Z 439.324,A -85,B 0,C 180,E1 -437.178,E2 -437.178} C_VEL
LIN {X 0,Y 608.538,Z 531,A -85,B 0,C 180,E1 -438.277,E2 -438.277} C_VEL
LIN {X 0,Y 608.514,Z 544.251,A -85,B 0,C 180,E1 -438.572,E2 -438.572} C_VEL
LIN {X 0,Y 608.517,Z 556.604,A -85,B 0,C 180,E1 -438.981,E2 -438.981} C_VEL
LIN {X 0,Y 608.498,Z 568.653,A -85,B 0,C 180,E1 -439.52,E2 -439.52} C_VEL
LIN {X 0,Y 608.48,Z 580.212,A -85,B 0,C 180,E1 -440.192,E2 -440.192} C_VEL
LIN {X 0,Y 608.485,Z 590.606,A -85,B 0,C 180,E1 -440.947,E2 -440.947} C_VEL
LIN {X 0,Y 608.474,Z 599.122,A -85,B 0,C 180,E1 -441.7,E2 -441.7} C_VEL
LIN {X 0,Y 608.47,Z 606.968,A -85,B 0,C 180,E1 -442.535,E2 -442.535} C_VEL
LIN {X 0,Y 608.46,Z 614.29,A -85,B 0,C 180,E1 -443.485,E2 -443.485} C_VEL
LIN {X 0,Y 608.45,Z 619.871,A -85,B 0,C 180,E1 -444.367,E2 -444.367} C_VEL
LIN {X 0,Y 608.432,Z 624.954,A -85,B 0,C 180,E1 -445.363,E2 -445.363} C_VEL
LIN {X 0,Y 608.449,Z 628.899,A -85,B 0,C 180,E1 -446.359,E2 -446.359} C_VEL
LIN {X 0,Y 608.425,Z 631.811,A -85,B 0,C 180,E1 -447.353,E2 -447.353} C_VEL
LIN {X 0,Y 608.442,Z 633.203,A -85,B 0,C 180,E1 -448.015,E2 -448.015} C_VEL
LIN {X 0,Y 608.438,Z 634.784,A -85,B 0,C 180,E1 -449.339,E2 -449.339} C_VEL
LIN {X 0,Y 608.434,Z 635,A -85,B 0,C 180,E1 -450.001,E2 -450.001} C_VEL
LIN {X 0,Y 608.448,Z 634.183,A -85,B 0,C 180,E1 -451.325,E2 -451.325} C_VEL
LIN {X 0,Y 608.443,Z 633.2,A -85,B 0,C 180,E1 -451.987,E2 -451.987} C_VEL
LIN {X 0,Y 608.425,Z 631.807,A -85,B 0,C 180,E1 -452.649,E2 -452.649} C_VEL
LIN {X 0,Y 608.449,Z 628.893,A -85,B 0,C 180,E1 -453.643,E2 -453.643} C_VEL
LIN {X 0,Y 608.432,Z 624.946,A -85,B 0,C 180,E1 -454.639,E2 -454.639} C_VEL
LIN {X 0,Y 608.437,Z 618.872,A -85,B 0,C 180,E1 -455.802,E2 -455.802} C_VEL
LIN {X 0,Y 608.463,Z 612.229,A -85,B 0,C 180,E1 -456.8,E2 -456.8} C_VEL
LIN {X 0,Y 608.456,Z 603.982,A -85,B 0,C 180,E1 -457.801,E2 -457.801} C_VEL
LIN {X 0,Y 608.472,Z 595.527,A -85,B 0,C 180,E1 -458.637,E2 -458.637} C_VEL
LIN {X 0,Y 608.471,Z 585.08,A -85,B 0,C 180,E1 -459.474,E2 -459.474} C_VEL
LIN {X 0,Y 608.494,Z 574.742,A -85,B 0,C 180,E1 -460.145,E2 -460.145} C_VEL
LIN {X 0,Y 608.521,Z 563.239,A -85,B 0,C 180,E1 -460.741,E2 -460.741} C_VEL
LIN {X 0,Y 608.531,Z 550.861,A -85,B 0,C 180,E1 -461.226,E2 -461.226} C_VEL
LIN {X 0,Y 608.537,Z 537.405,A -85,B 0,C 180,E1 -461.598,E2 -461.598} C_VEL
LIN {X 0,Y 608.547,Z 525.024,A -85,B 0,C 180,E1 -461.809,E2 -461.809} C_VEL
LIN {X 0,Y 608.496,Z 423.077,A -85,B 0,C 180,E1 -463.017,E2 -463.017} C_VEL
LIN {X 0,Y 608.498,Z 401.536,A -85,B 0,C 180,E1 -465.921,E2 -465.921} C_VEL
LIN {X 0,Y 608.505,Z 382.808,A -85,B 0,C 180,E1 -468.497,E2 -468.497} C_VEL
LIN {X 0,Y 608.57,Z 363.756,A -85,B 0,C 180,E1 -471.155,E2 -471.155} C_VEL
LIN {X 0,Y 608.452,Z 355.69,A -85,B 0,C 180,E1 -472.317,E2 -472.317} C_VEL
LIN {X 0,Y 608.453,Z 355.688,A -85,B 0,C 180,E1 -474.572,E2 -474.572} C_VEL
LIN {X 0,Y 608.486,Z 355.691,A -85,B 0,C 180,E1 -477.208,E2 -477.208} C_VEL
LIN {X 0,Y 608.472,Z 355.686,A -85,B 0,C 180,E1 -479.972,E2 -479.972} C_VEL
LIN {X 0,Y 608.456,Z 355.688,A -85,B 0,C 180,E1 -482.521,E2 -482.521} C_VEL
LIN {X 0,Y 608.452,Z 355.697,A -85,B 0,C 180,E1 -485.278,E2 -485.278} C_VEL
LIN {X 0,Y 608.472,Z 355.687,A -85,B 0,C 180,E1 -487.747,E2 -487.747} C_VEL
LIN {X 0,Y 608.445,Z 355.689,A -85,B 0,C 180,E1 -490.328,E2 -490.328} C_VEL
LIN {X 0,Y 608.478,Z 355.69,A -85,B 0,C 180,E1 -493.309,E2 -493.309} C_VEL
LIN {X 0,Y 608.47,Z 355.686,A -85,B 0,C 180,E1 -496.13,E2 -496.13} C_VEL
LIN {X 0,Y 608.455,Z 355.696,A -85,B 0,C 180,E1 -498.823,E2 -498.823} C_VEL
LIN {X 0,Y 608.466,Z 355.686,A -85,B 0,C 180,E1 -501.761,E2 -501.761} C_VEL
LIN {X 0,Y 608.448,Z 355.688,A -85,B 0,C 180,E1 -503.955,E2 -503.955} C_VEL
LIN {X 0,Y 608.451,Z 355.691,A -85,B 0,C 180,E1 -506.328,E2 -506.328} C_VEL
LIN {X 0,Y 608.45,Z 355.698,A -85,B 0,C 180,E1 -508.733,E2 -508.733} C_VEL
LIN {X 0,Y 608.474,Z 355.686,A -85,B 0,C 180,E1 -511.381,E2 -511.381} C_VEL
LIN {X 0,Y 608.445,Z 355.69,A -85,B 0,C 180,E1 -513.964,E2 -513.964} C_VEL
LIN {X 0,Y 608.462,Z 355.69,A -85,B 0,C 180,E1 -516.155,E2 -516.155} C_VEL
LIN {X 0,Y 608.474,Z 355.692,A -85,B 0,C 180,E1 -518.309,E2 -518.309} C_VEL
LIN {X 0,Y 608.472,Z 355.685,A -85,B 0,C 180,E1 -521.285,E2 -521.285} C_VEL
LIN {X 0,Y 608.457,Z 355.69,A -85,B 0,C 180,E1 -523.906,E2 -523.906} C_VEL
LIN {X 0,Y 608.461,Z 355.692,A -85,B 0,C 180,E1 -526.644,E2 -526.644} C_VEL
LIN {X 0,Y 608.466,Z 355.686,A -85,B 0,C 180,E1 -529.35,E2 -529.35} C_VEL
LIN {X 0,Y 608.482,Z 355.691,A -85,B 0,C 180,E1 -532.033,E2 -532.033} C_VEL
LIN {X 0,Y 608.465,Z 355.689,A -85,B 0,C 180,E1 -534.698,E2 -534.698} C_VEL
LIN {X 0,Y 608.481,Z 355.684,A -85,B 0,C 180,E1 -537.352,E2 -537.352} C_VEL
LIN {X 0,Y 608.482,Z 355.693,A -85,B 0,C 180,E1 -540,E2 -540} C_VEL
LIN {X 0,Y 608.481,Z 355.685,A -85,B 0,C 180,E1 -542.648,E2 -542.648} C_VEL
LIN {X 0,Y 608.465,Z 355.687,A -85,B 0,C 180,E1 -545.302,E2 -545.302} C_VEL
LIN {X 0,Y 608.484,Z 355.693,A -85,B 0,C 180,E1 -547.967,E2 -547.967} C_VEL
LIN {X 0,Y 608.46,Z 355.689,A -85,B 0,C 180,E1 -549.458,E2 -549.458} C_VEL
LIN {X 0,Y 607.788,Z 355.779,A -85,B 0,C 180,E1 -550.01,E2 -550.01} C_VEL
LIN {X 0,Y 604.937,Z 356.134,A -85,B 0,C 180,E1 -550.907,E2 -550.907} C_VEL
LIN {X 0,Y 602.531,Z 356.433,A -85,B 0,C 180,E1 -551.629,E2 -551.629} C_VEL
LIN {X 0,Y 601.498,Z 356.559,A -85,B 0,C 180,E1 -552.186,E2 -552.186} C_VEL
LIN {X 0,Y 601.413,Z 356.567,A -85,B 0,C 180,E1 -552.374,E2 -552.374} C_VEL
LIN {X 0,Y 601.433,Z 356.562,A -85,B 0,C 180,E1 -554.897,E2 -554.897} C_VEL
LIN {X 0,Y 601.435,Z 356.563,A -85,B 0,C 180,E1 -556.986,E2 -556.986} C_VEL
LIN {X 0,Y 601.409,Z 356.573,A -85,B 0,C 180,E1 -559.809,E2 -559.809} C_VEL
LIN {X 0,Y 601.417,Z 356.564,A -85,B 0,C 180,E1 -562.683,E2 -562.683} C_VEL
LIN {X 0,Y 601.404,Z 356.567,A -85,B 0,C 180,E1 -564.879,E2 -564.879} C_VEL
LIN {X 0,Y 601.415,Z 356.572,A -85,B 0,C 180,E1 -567.361,E2 -567.361} C_VEL
LIN {X 0,Y 601.433,Z 356.563,A -85,B 0,C 180,E1 -570.164,E2 -570.164} C_VEL
LIN {X 0,Y 601.462,Z 356.727,A -85,B 0,C 180,E1 -572.653,E2 -572.653} C_VEL
LIN {X 0,Y 601.475,Z 373.107,A -85,B 0,C 180,E1 -575.403,E2 -575.403} C_VEL
LIN {X 0,Y 601.417,Z 390.435,A -85,B 0,C 180,E1 -578.269,E2 -578.269} C_VEL
LIN {X 0,Y 601.427,Z 394.156,A -85,B 0,C 180,E1 -578.88,E2 -578.88} C_VEL
LIN {X 0,Y 601.66,Z 400.938,A -85,B 0,C 180,E1 -578.972,E2 -578.972} C_VEL
LIN {X 0,Y 601.617,Z 501.224,A -85,B 0,C 180,E1 -580.19,E2 -580.19} C_VEL
LIN {X 0,Y 601.569,Z 514.526,A -85,B 0,C 180,E1 -580.491,E2 -580.491} C_VEL
LIN {X 0,Y 601.555,Z 527.176,A -85,B 0,C 180,E1 -580.919,E2 -580.919} C_VEL
LIN {X 0,Y 601.516,Z 538.844,A -85,B 0,C 180,E1 -581.452,E2 -581.452} C_VEL
LIN {X 0,Y 601.498,Z 549.836,A -85,B 0,C 180,E1 -582.097,E2 -582.097} C_VEL
LIN {X 0,Y 601.432,Z 560.764,A -85,B 0,C 180,E1 -582.897,E2 -582.897} C_VEL
LIN {X 0,Y 601.419,Z 569.701,A -85,B 0,C 180,E1 -583.703,E2 -583.703} C_VEL
LIN {X 0,Y 601.393,Z 578.075,A -85,B 0,C 180,E1 -584.627,E2 -584.627} C_VEL
LIN {X 0,Y 601.376,Z 586.009,A -85,B 0,C 180,E1 -585.711,E2 -585.711} C_VEL
LIN {X 0,Y 601.36,Z 592.719,A -85,B 0,C 180,E1 -586.881,E2 -586.881} C_VEL
LIN {X 0,Y 601.36,Z 596.934,A -85,B 0,C 180,E1 -587.824,E2 -587.824} C_VEL
LIN {X 0,Y 601.332,Z 600.184,A -85,B 0,C 180,E1 -588.767,E2 -588.767} C_VEL
LIN {X 0,Y 601.306,Z 603.136,A -85,B 0,C 180,E1 -589.996,E2 -589.996} C_VEL
LIN {X 0,Y 601.314,Z 604.369,A -85,B 0,C 180,E1 -590.865,E2 -590.865} C_VEL
LIN {X 0,Y 601.327,Z 604.932,A -85,B 0,C 180,E1 -591.724,E2 -591.724} C_VEL
LIN {X 0,Y 601.334,Z 604.842,A -85,B 0,C 180,E1 -592.631,E2 -592.631} C_VEL
LIN {X 0,Y 601.318,Z 603.699,A -85,B 0,C 180,E1 -593.751,E2 -593.751} C_VEL
LIN {X 0,Y 601.339,Z 600.92,A -85,B 0,C 180,E1 -595.062,E2 -595.062} C_VEL
LIN {X 0,Y 601.34,Z 597.634,A -85,B 0,C 180,E1 -596.078,E2 -596.078} C_VEL
LIN {X 0,Y 601.362,Z 592.296,A -85,B 0,C 180,E1 -597.294,E2 -597.294} C_VEL
LIN {X 0,Y 601.372,Z 586.72,A -85,B 0,C 180,E1 -598.271,E2 -598.271} C_VEL
LIN {X 0,Y 601.408,Z 579.776,A -85,B 0,C 180,E1 -599.252,E2 -599.252} C_VEL
LIN {X 0,Y 601.412,Z 571.315,A -85,B 0,C 180,E1 -600.221,E2 -600.221} C_VEL
LIN {X 0,Y 601.441,Z 561.819,A -85,B 0,C 180,E1 -601.107,E2 -601.107} C_VEL
LIN {X 0,Y 601.455,Z 552.013,A -85,B 0,C 180,E1 -601.849,E2 -601.849} C_VEL
LIN {X 0,Y 601.487,Z 540.412,A -85,B 0,C 180,E1 -602.554,E2 -602.554} C_VEL
LIN {X 0,Y 601.527,Z 528.301,A -85,B 0,C 180,E1 -603.127,E2 -603.127} C_VEL
LIN {X 0,Y 601.575,Z 515.423,A -85,B 0,C 180,E1 -603.574,E2 -603.574} C_VEL
LIN {X 0,Y 601.62,Z 502.201,A -85,B 0,C 180,E1 -603.882,E2 -603.882} C_VEL
LIN {X 0,Y 601.64,Z 463.414,A -85,B 0,C 180,E1 -604.369,E2 -604.369} C_VEL
LIN {X 0,Y 601.557,Z 395.16,A -85,B 0,C 180,E1 -605.189,E2 -605.189} C_VEL
LIN {X 0,Y 601.423,Z 394.195,A -85,B 0,C 180,E1 -605.204,E2 -605.204} C_VEL
LIN {X 0,Y 601.462,Z 376.986,A -85,B 0,C 180,E1 -608.042,E2 -608.042} C_VEL
LIN {X 0,Y 601.534,Z 359.868,A -85,B 0,C 180,E1 -610.904,E2 -610.904} C_VEL
LIN {X 0,Y 601.433,Z 356.565,A -85,B 0,C 180,E1 -611.493,E2 -611.493} C_VEL
LIN {X 0,Y 601.42,Z 356.571,A -85,B 0,C 180,E1 -614.408,E2 -614.408} C_VEL
LIN {X 0,Y 601.42,Z 356.565,A -85,B 0,C 180,E1 -617.171,E2 -617.171} C_VEL
LIN {X 0,Y 601.438,Z 356.563,A -85,B 0,C 180,E1 -619.904,E2 -619.904} C_VEL
LIN {X 0,Y 601.448,Z 356.568,A -85,B 0,C 180,E1 -622.614,E2 -622.614} C_VEL
LIN {X 0,Y 601.418,Z 356.564,A -85,B 0,C 180,E1 -625.307,E2 -625.307} C_VEL
LIN {X 0,Y 601.437,Z 356.566,A -85,B 0,C 180,E1 -627.99,E2 -627.99} C_VEL
LIN {X 0,Y 601.453,Z 356.564,A -85,B 0,C 180,E1 -630.669,E2 -630.669} C_VEL
LIN {X 0,Y 601.427,Z 356.563,A -85,B 0,C 180,E1 -633.349,E2 -633.349} C_VEL
LIN {X 0,Y 601.417,Z 356.571,A -85,B 0,C 180,E1 -636.036,E2 -636.036} C_VEL
LIN {X 0,Y 601.412,Z 356.566,A -85,B 0,C 180,E1 -638.737,E2 -638.737} C_VEL
LIN {X 0,Y 601.435,Z 356.563,A -85,B 0,C 180,E1 -641.457,E2 -641.457} C_VEL
LIN {X 0,Y 601.422,Z 356.571,A -85,B 0,C 180,E1 -644.204,E2 -644.204} C_VEL
LIN {X 0,Y 601.421,Z 356.563,A -85,B 0,C 180,E1 -646.985,E2 -646.985} C_VEL
LIN {X 0,Y 601.402,Z 356.574,A -85,B 0,C 180,E1 -649.808,E2 -649.808} C_VEL
LIN {X 0,Y 601.412,Z 356.565,A -85,B 0,C 180,E1 -652.682,E2 -652.682} C_VEL
LIN {X 0,Y 601.401,Z 356.566,A -85,B 0,C 180,E1 -654.877,E2 -654.877} C_VEL
LIN {X 0,Y 601.417,Z 356.573,A -85,B 0,C 180,E1 -657.866,E2 -657.866} C_VEL
LIN {X 0,Y 601.447,Z 356.564,A -85,B 0,C 180,E1 -660.162,E2 -660.162} C_VEL
LIN {X 0,Y 601.416,Z 356.564,A -85,B 0,C 180,E1 -662.714,E2 -662.714} C_VEL
LIN {X 0,Y 601.42,Z 356.566,A -85,B 0,C 180,E1 -665.115,E2 -665.115} C_VEL
LIN {X 0,Y 601.431,Z 356.569,A -85,B 0,C 180,E1 -667.418,E2 -667.418} C_VEL
LIN {X 0,Y 601.408,Z 356.569,A -85,B 0,C 180,E1 -669.994,E2 -669.994} C_VEL
LIN {X 0,Y 601.407,Z 356.565,A -85,B 0,C 180,E1 -672.669,E2 -672.669} C_VEL
LIN {X 0,Y 601.42,Z 356.574,A -85,B 0,C 180,E1 -675.481,E2 -675.481} C_VEL
LIN {X 0,Y 601.428,Z 356.565,A -85,B 0,C 180,E1 -678.405,E2 -678.405} C_VEL
LIN {X 0,Y 601.443,Z 356.609,A -85,B 0,C 180,E1 -678.632,E2 -678.632} C_VEL
LIN {X 0,Y 601.472,Z 369.959,A -85,B 0,C 180,E1 -680.878,E2 -680.878} C_VEL
LIN {X 0,Y 601.472,Z 385.284,A -85,B 0,C 180,E1 -683.422,E2 -683.422} C_VEL
LIN {X 0,Y 601.405,Z 394.19,A -85,B 0,C 180,E1 -684.885,E2 -684.885} C_VEL
LIN {X 0,Y 601.664,Z 402.261,A -85,B 0,C 180,E1 -684.988,E2 -684.988} C_VEL
LIN {X 0,Y 601.588,Z 501.505,A -85,B 0,C 180,E1 -686.194,E2 -686.194} C_VEL
LIN {X 0,Y 601.576,Z 515.558,A -85,B 0,C 180,E1 -686.52,E2 -686.52} C_VEL
LIN {X 0,Y 601.536,Z 528.192,A -85,B 0,C 180,E1 -686.96,E2 -686.96} C_VEL
LIN {X 0,Y 601.499,Z 539.508,A -85,B 0,C 180,E1 -687.488,E2 -687.488} C_VEL
LIN {X 0,Y 601.456,Z 551.06,A -85,B 0,C 180,E1 -688.178,E2 -688.178} C_VEL
LIN {X 0,Y 601.452,Z 561.723,A -85,B 0,C 180,E1 -688.975,E2 -688.975} C_VEL
LIN {X 0,Y 601.399,Z 571.156,A -85,B 0,C 180,E1 -689.854,E2 -689.854} C_VEL
LIN {X 0,Y 601.37,Z 579.232,A -85,B 0,C 180,E1 -690.772,E2 -690.772} C_VEL
LIN {X 0,Y 601.376,Z 586.267,A -85,B 0,C 180,E1 -691.751,E2 -691.751} C_VEL
LIN {X 0,Y 601.34,Z 592.726,A -85,B 0,C 180,E1 -692.883,E2 -692.883} C_VEL
LIN {X 0,Y 601.381,Z 596.147,A -85,B 0,C 180,E1 -693.635,E2 -693.635} C_VEL
LIN {X 0,Y 601.336,Z 600.128,A -85,B 0,C 180,E1 -694.749,E2 -694.749} C_VEL
LIN {X 0,Y 601.348,Z 602.871,A -85,B 0,C 180,E1 -695.855,E2 -695.855} C_VEL
LIN {X 0,Y 601.324,Z 604.046,A -85,B 0,C 180,E1 -696.586,E2 -696.586} C_VEL
LIN {X 0,Y 601.34,Z 604.806,A -85,B 0,C 180,E1 -697.409,E2 -697.409} C_VEL
LIN {X 0,Y 601.332,Z 604.99,A -85,B 0,C 180,E1 -698.038,E2 -698.038} C_VEL
LIN {X 0,Y 601.337,Z 604.375,A -85,B 0,C 180,E1 -699.222,E2 -699.222} C_VEL
LIN {X 0,Y 601.315,Z 602.966,A -85,B 0,C 180,E1 -700.187,E2 -700.187} C_VEL
LIN {X 0,Y 601.342,Z 600.553,A -85,B 0,C 180,E1 -701.198,E2 -701.198} C_VEL
LIN {X 0,Y 601.346,Z 596.76,A -85,B 0,C 180,E1 -702.31,E2 -702.31} C_VEL
LIN {X 0,Y 601.36,Z 591.76,A -85,B 0,C 180,E1 -703.395,E2 -703.395} C_VEL
LIN {X 0,Y 601.356,Z 585.817,A -85,B 0,C 180,E1 -704.407,E2 -704.407} C_VEL
LIN {X 0,Y 601.398,Z 578.179,A -85,B 0,C 180,E1 -705.448,E2 -705.448} C_VEL
LIN {X 0,Y 601.421,Z 570.098,A -85,B 0,C 180,E1 -706.346,E2 -706.346} C_VEL
LIN {X 0,Y 601.461,Z 559.94,A -85,B 0,C 180,E1 -707.258,E2 -707.258} C_VEL
LIN {X 0,Y 601.468,Z 549.294,A -85,B 0,C 180,E1 -708.03,E2 -708.03} C_VEL
LIN {X 0,Y 601.513,Z 537.672,A -85,B 0,C 180,E1 -708.698,E2 -708.698} C_VEL
LIN {X 0,Y 601.552,Z 524.619,A -85,B 0,C 180,E1 -709.269,E2 -709.269} C_VEL
LIN {X 0,Y 601.591,Z 511.792,A -85,B 0,C 180,E1 -709.674,E2 -709.674} C_VEL
LIN {X 0,Y 601.603,Z 499.448,A -85,B 0,C 180,E1 -709.929,E2 -709.929} C_VEL
LIN {X 0,Y 601.559,Z 395.108,A -85,B 0,C 180,E1 -711.19,E2 -711.19} C_VEL
LIN {X 0,Y 601.432,Z 394.098,A -85,B 0,C 180,E1 -711.22,E2 -711.22} C_VEL
LIN {X 0,Y 601.483,Z 377.455,A -85,B 0,C 180,E1 -713.964,E2 -713.964} C_VEL
LIN {X 0,Y 601.528,Z 361.371,A -85,B 0,C 180,E1 -716.651,E2 -716.651} C_VEL
LIN {X 0,Y 601.443,Z 356.564,A -85,B 0,C 180,E1 -717.488,E2 -717.488} C_VEL
LIN {X 0,Y 601.436,Z 356.564,A -85,B 0,C 180,E1 -720,E2 -720} C_VEL
LIN {X 0,Y 601.446,Z 356.569,A -85,B 0,C 180,E1 -722.679,E2 -722.679} C_VEL
LIN {X 0,Y 601.425,Z 356.563,A -85,B 0,C 180,E1 -725.364,E2 -725.364} C_VEL
LIN {X 0,Y 601.435,Z 356.567,A -85,B 0,C 180,E1 -728.061,E2 -728.061} C_VEL
LIN {X 0,Y 601.42,Z 356.565,A -85,B 0,C 180,E1 -731.017,E2 -731.017} C_VEL
LIN {X 0,Y 601.414,Z 356.566,A -85,B 0,C 180,E1 -733.516,E2 -733.516} C_VEL
LIN {X 0,Y 601.451,Z 356.567,A -85,B 0,C 180,E1 -736.287,E2 -736.287} C_VEL
LIN {X 0,Y 601.413,Z 356.565,A -85,B 0,C 180,E1 -739.099,E2 -739.099} C_VEL
LIN {X 0,Y 601.407,Z 356.566,A -85,B 0,C 180,E1 -741.239,E2 -741.239} C_VEL
LIN {X 0,Y 601.42,Z 356.567,A -85,B 0,C 180,E1 -743.41,E2 -743.41} C_VEL
LIN {X 0,Y 601.405,Z 356.568,A -85,B 0,C 180,E1 -746.364,E2 -746.364} C_VEL
LIN {X 0,Y 601.436,Z 356.562,A -85,B 0,C 180,E1 -748.791,E2 -748.791} C_VEL
LIN {X 0,Y 601.436,Z 356.569,A -85,B 0,C 180,E1 -751.46,E2 -751.46} C_VEL
LIN {X 0,Y 601.427,Z 356.565,A -85,B 0,C 180,E1 -754.119,E2 -754.119} C_VEL
LIN {X 0,Y 601.406,Z 356.566,A -85,B 0,C 180,E1 -756.583,E2 -756.583} C_VEL
LIN {X 0,Y 601.432,Z 356.57,A -85,B 0,C 180,E1 -759.537,E2 -759.537} C_VEL
LIN {X 0,Y 601.433,Z 356.563,A -85,B 0,C 180,E1 -762.595,E2 -762.595} C_VEL
LIN {X 0,Y 601.419,Z 356.57,A -85,B 0,C 180,E1 -765.483,E2 -765.483} C_VEL
LIN {X 0,Y 601.419,Z 356.565,A -85,B 0,C 180,E1 -768.408,E2 -768.408} C_VEL
LIN {X 0,Y 601.435,Z 356.569,A -85,B 0,C 180,E1 -770.877,E2 -770.877} C_VEL
LIN {X 0,Y 601.441,Z 356.562,A -85,B 0,C 180,E1 -773.735,E2 -773.735} C_VEL
LIN {X 0,Y 601.432,Z 356.563,A -85,B 0,C 180,E1 -776.065,E2 -776.065} C_VEL
LIN {X 0,Y 601.431,Z 356.569,A -85,B 0,C 180,E1 -779.06,E2 -779.06} C_VEL
LIN {X 0,Y 601.429,Z 356.564,A -85,B 0,C 180,E1 -781.374,E2 -781.374} C_VEL
LIN {X 0,Y 601.404,Z 356.566,A -85,B 0,C 180,E1 -783.638,E2 -783.638} C_VEL
LIN {X 0,Y 601.424,Z 356.574,A -85,B 0,C 180,E1 -786.591,E2 -786.591} C_VEL
LIN {X 0,Y 601.474,Z 356.768,A -85,B 0,C 180,E1 -787.582,E2 -787.582} C_VEL
LIN {X 0,Y 601.623,Z 366.952,A -85,B 0,C 180,E1 -789.044,E2 -789.044} C_VEL
LIN {X 0,Y 601.562,Z 387.696,A -85,B 0,C 180,E1 -791.966,E2 -791.966} C_VEL
LIN {X 0,Y 601.483,Z 407.845,A -85,B 0,C 180,E1 -794.759,E2 -794.759} C_VEL
LIN {X 0,Y 601.46,Z 422.8,A -85,B 0,C 180,E1 -796.809,E2 -796.809} C_VEL
LIN {X 0,Y 601.674,Z 428.592,A -85,B 0,C 180,E1 -796.899,E2 -796.899} C_VEL
LIN {X 0,Y 601.604,Z 531,A -85,B 0,C 180,E1 -798.14,E2 -798.14} C_VEL
LIN {X 0,Y 601.573,Z 544.252,A -85,B 0,C 180,E1 -798.439,E2 -798.439} C_VEL
LIN {X 0,Y 601.543,Z 555.979,A -85,B 0,C 180,E1 -798.828,E2 -798.828} C_VEL
LIN {X 0,Y 601.515,Z 566.943,A -85,B 0,C 180,E1 -799.312,E2 -799.312} C_VEL
LIN {X 0,Y 601.479,Z 577.596,A -85,B 0,C 180,E1 -799.907,E2 -799.907} C_VEL
LIN {X 0,Y 601.446,Z 588.488,A -85,B 0,C 180,E1 -800.67,E2 -800.67} C_VEL
LIN {X 0,Y 601.429,Z 599.122,A -85,B 0,C 180,E1 -801.602,E2 -801.602} C_VEL
LIN {X 0,Y 601.417,Z 606.968,A -85,B 0,C 180,E1 -802.447,E2 -802.447} C_VEL
LIN {X 0,Y 601.369,Z 614.229,A -85,B 0,C 180,E1 -803.399,E2 -803.399} C_VEL
LIN {X 0,Y 601.371,Z 619.871,A -85,B 0,C 180,E1 -804.3,E2 -804.3} C_VEL
LIN {X 0,Y 601.337,Z 624.954,A -85,B 0,C 180,E1 -805.308,E2 -805.308} C_VEL
LIN {X 0,Y 601.367,Z 628.899,A -85,B 0,C 180,E1 -806.316,E2 -806.316} C_VEL
LIN {X 0,Y 601.325,Z 631.811,A -85,B 0,C 180,E1 -807.321,E2 -807.321} C_VEL
LIN {X 0,Y 601.341,Z 633.203,A -85,B 0,C 180,E1 -807.992,E2 -807.992} C_VEL
LIN {X 0,Y 601.339,Z 634.784,A -85,B 0,C 180,E1 -809.331,E2 -809.331} C_VEL
LIN {X 0,Y 601.335,Z 635,A -85,B 0,C 180,E1 -810.001,E2 -810.001} C_VEL
LIN {X 0,Y 601.348,Z 634.183,A -85,B 0,C 180,E1 -811.34,E2 -811.34} C_VEL
LIN {X 0,Y 601.342,Z 633.201,A -85,B 0,C 180,E1 -812.01,E2 -812.01} C_VEL
LIN {X 0,Y 601.325,Z 631.807,A -85,B 0,C 180,E1 -812.68,E2 -812.68} C_VEL
LIN {X 0,Y 601.367,Z 628.893,A -85,B 0,C 180,E1 -813.686,E2 -813.686} C_VEL
LIN {X 0,Y 601.337,Z 624.946,A -85,B 0,C 180,E1 -814.694,E2 -814.694} C_VEL
LIN {X 0,Y 601.372,Z 618.872,A -85,B 0,C 180,E1 -815.87,E2 -815.87} C_VEL
LIN {X 0,Y 601.382,Z 612.229,A -85,B 0,C 180,E1 -816.881,E2 -816.881} C_VEL
LIN {X 0,Y 601.401,Z 603.982,A -85,B 0,C 180,E1 -817.893,E2 -817.893} C_VEL
LIN {X 0,Y 601.436,Z 595.528,A -85,B 0,C 180,E1 -818.738,E2 -818.738} C_VEL
LIN {X 0,Y 601.442,Z 585.081,A -85,B 0,C 180,E1 -819.586,E2 -819.586} C_VEL
LIN {X 0,Y 601.472,Z 574.744,A -85,B 0,C 180,E1 -820.265,E2 -820.265} C_VEL
LIN {X 0,Y 601.536,Z 563.893,A -85,B 0,C 180,E1 -820.836,E2 -820.836} C_VEL
LIN {X 0,Y 601.557,Z 551.357,A -85,B 0,C 180,E1 -821.341,E2 -821.341} C_VEL
LIN {X 0,Y 601.569,Z 538.318,A -85,B 0,C 180,E1 -821.713,E2 -821.713} C_VEL
LIN {X 0,Y 601.614,Z 525.024,A -85,B 0,C 180,E1 -821.947,E2 -821.947} C_VEL
LIN {X 0,Y 601.572,Z 423.748,A -85,B 0,C 180,E1 -823.161,E2 -823.161} C_VEL
LIN {X 0,Y 601.459,Z 422.787,A -85,B 0,C 180,E1 -823.193,E2 -823.193} C_VEL
LIN {X 0,Y 601.489,Z 402.795,A -85,B 0,C 180,E1 -825.938,E2 -825.938} C_VEL
LIN {X 0,Y 601.533,Z 385.164,A -85,B 0,C 180,E1 -828.389,E2 -828.389} C_VEL
LIN {X 0,Y 601.641,Z 366.771,A -85,B 0,C 180,E1 -830.981,E2 -830.981} C_VEL
LIN {X 0,Y 601.472,Z 356.759,A -85,B 0,C 180,E1 -832.42,E2 -832.42} C_VEL
LIN {X 0,Y 601.407,Z 356.568,A -85,B 0,C 180,E1 -834.879,E2 -834.879} C_VEL
LIN {X 0,Y 601.423,Z 356.574,A -85,B 0,C 180,E1 -837.363,E2 -837.363} C_VEL
LIN {X 0,Y 601.434,Z 356.562,A -85,B 0,C 180,E1 -840.164,E2 -840.164} C_VEL
LIN {X 0,Y 601.421,Z 356.566,A -85,B 0,C 180,E1 -842.715,E2 -842.715} C_VEL
LIN {X 0,Y 601.421,Z 356.573,A -85,B 0,C 180,E1 -845.115,E2 -845.115} C_VEL
LIN {X 0,Y 601.441,Z 356.567,A -85,B 0,C 180,E1 -847.419,E2 -847.419} C_VEL
LIN {X 0,Y 601.417,Z 356.564,A -85,B 0,C 180,E1 -849.995,E2 -849.995} C_VEL
LIN {X 0,Y 601.414,Z 356.569,A -85,B 0,C 180,E1 -852.671,E2 -852.671} C_VEL
LIN {X 0,Y 601.432,Z 356.565,A -85,B 0,C 180,E1 -855.482,E2 -855.482} C_VEL
LIN {X 0,Y 601.426,Z 356.565,A -85,B 0,C 180,E1 -858.407,E2 -858.407} C_VEL
LIN {X 0,Y 601.411,Z 356.575,A -85,B 0,C 180,E1 -860.873,E2 -860.873} C_VEL
LIN {X 0,Y 601.401,Z 356.568,A -85,B 0,C 180,E1 -863.417,E2 -863.417} C_VEL
LIN {X 0,Y 601.436,Z 356.562,A -85,B 0,C 180,E1 -866.065,E2 -866.065} C_VEL
LIN {X 0,Y 601.423,Z 356.571,A -85,B 0,C 180,E1 -868.546,E2 -868.546} C_VEL
LIN {X 0,Y 601.433,Z 356.563,A -85,B 0,C 180,E1 -871.373,E2 -871.373} C_VEL
LIN {X 0,Y 601.403,Z 356.565,A -85,B 0,C 180,E1 -873.636,E2 -873.636} C_VEL
LIN {X 0,Y 601.417,Z 356.574,A -85,B 0,C 180,E1 -876.59,E2 -876.59} C_VEL
LIN {X 0,Y 601.431,Z 356.562,A -85,B 0,C 180,E1 -879.478,E2 -879.478} C_VEL
LIN {X 0,Y 601.398,Z 356.574,A -85,B 0,C 180,E1 -882.312,E2 -882.312} C_VEL
LIN {X 0,Y 601.413,Z 356.575,A -85,B 0,C 180,E1 -884.409,E2 -884.409} C_VEL
LIN {X 0,Y 601.42,Z 356.564,A -85,B 0,C 180,E1 -887.172,E2 -887.172} C_VEL
LIN {X 0,Y 601.44,Z 356.565,A -85,B 0,C 180,E1 -889.905,E2 -889.905} C_VEL
LIN {X 0,Y 601.443,Z 356.564,A -85,B 0,C 180,E1 -892.615,E2 -892.615} C_VEL
LIN {X 0,Y 601.428,Z 356.563,A -85,B 0,C 180,E1 -895.308,E2 -895.308} C_VEL
LIN {X 0,Y 601.435,Z 356.57,A -85,B 0,C 180,E1 -897.991,E2 -897.991} C_VEL
LIN {X 0,Y 601.45,Z 356.561,A -85,B 0,C 180,E1 -900.67,E2 -900.67} C_VEL
LIN {X 0,Y 601.431,Z 356.564,A -85,B 0,C 180,E1 -903.35,E2 -903.35} C_VEL
LIN {X 0,Y 601.423,Z 356.572,A -85,B 0,C 180,E1 -906.037,E2 -906.037} C_VEL
LIN {X 0,Y 601.417,Z 356.564,A -85,B 0,C 180,E1 -908.738,E2 -908.738} C_VEL
LIN {X 0,Y 601.438,Z 356.566,A -85,B 0,C 180,E1 -911.458,E2 -911.458} C_VEL
LIN {X 0,Y 601.413,Z 356.567,A -85,B 0,C 180,E1 -912.374,E2 -912.374} C_VEL
LIN {X 0,Y 600.745,Z 356.65,A -85,B 0,C 180,E1 -912.933,E2 -912.933} C_VEL
LIN {X 0,Y 597.896,Z 357.012,A -85,B 0,C 180,E1 -913.841,E2 -913.841} C_VEL
LIN {X 0,Y 595.487,Z 357.307,A -85,B 0,C 180,E1 -914.571,E2 -914.571} C_VEL
LIN {X 0,Y 594.451,Z 357.434,A -85,B 0,C 180,E1 -915.135,E2 -915.135} C_VEL
LIN {X 0,Y 594.365,Z 357.446,A -85,B 0,C 180,E1 -915.326,E2 -915.326} C_VEL
LIN {X 0,Y 594.393,Z 357.442,A -85,B 0,C 180,E1 -917.193,E2 -917.193} C_VEL
LIN {X 0,Y 594.378,Z 357.445,A -85,B 0,C 180,E1 -920.054,E2 -920.054} C_VEL
LIN {X 0,Y 594.368,Z 357.444,A -85,B 0,C 180,E1 -922.967,E2 -922.967} C_VEL
LIN {X 0,Y 594.38,Z 357.445,A -85,B 0,C 180,E1 -925.193,E2 -925.193} C_VEL
LIN {X 0,Y 594.373,Z 357.452,A -85,B 0,C 180,E1 -927.523,E2 -927.523} C_VEL
LIN {X 0,Y 594.391,Z 357.44,A -85,B 0,C 180,E1 -930.328,E2 -930.328} C_VEL
LIN {X 0,Y 594.421,Z 357.459,A -85,B 0,C 180,E1 -932.539,E2 -932.539} C_VEL
LIN {X 0,Y 594.467,Z 371.651,A -85,B 0,C 180,E1 -934.955,E2 -934.955} C_VEL
LIN {X 0,Y 594.403,Z 387.474,A -85,B 0,C 180,E1 -937.609,E2 -937.609} C_VEL
LIN {X 0,Y 594.363,Z 394.199,A -85,B 0,C 180,E1 -938.727,E2 -938.727} C_VEL
LIN {X 0,Y 594.778,Z 398.48,A -85,B 0,C 180,E1 -938.788,E2 -938.788} C_VEL
LIN {X 0,Y 594.68,Z 501.642,A -85,B 0,C 180,E1 -940.057,E2 -940.057} C_VEL
LIN {X 0,Y 594.603,Z 514.96,A -85,B 0,C 180,E1 -940.366,E2 -940.366} C_VEL
LIN {X 0,Y 594.582,Z 526.832,A -85,B 0,C 180,E1 -940.773,E2 -940.773} C_VEL
LIN {X 0,Y 594.517,Z 538.02,A -85,B 0,C 180,E1 -941.283,E2 -941.283} C_VEL
LIN {X 0,Y 594.49,Z 549.022,A -85,B 0,C 180,E1 -941.923,E2 -941.923} C_VEL
LIN {X 0,Y 594.401,Z 560.517,A -85,B 0,C 180,E1 -942.768,E2 -942.768} C_VEL
LIN {X 0,Y 594.385,Z 570.649,A -85,B 0,C 180,E1 -943.701,E2 -943.701} C_VEL
LIN {X 0,Y 594.314,Z 579.076,A -85,B 0,C 180,E1 -944.664,E2 -944.664} C_VEL
LIN {X 0,Y 594.31,Z 586.789,A -85,B 0,C 180,E1 -945.756,E2 -945.756} C_VEL
LIN {X 0,Y 594.277,Z 593.339,A -85,B 0,C 180,E1 -946.95,E2 -946.95} C_VEL
LIN {X 0,Y 594.274,Z 598.362,A -85,B 0,C 180,E1 -948.164,E2 -948.164} C_VEL
LIN {X 0,Y 594.254,Z 602.014,A -85,B 0,C 180,E1 -949.423,E2 -949.423} C_VEL
LIN {X 0,Y 594.207,Z 603.678,A -85,B 0,C 180,E1 -950.305,E2 -950.305} C_VEL
LIN {X 0,Y 594.207,Z 604.749,A -85,B 0,C 180,E1 -951.317,E2 -951.317} C_VEL
LIN {X 0,Y 594.229,Z 604.922,A -85,B 0,C 180,E1 -952.412,E2 -952.412} C_VEL
LIN {X 0,Y 594.235,Z 603.739,A -85,B 0,C 180,E1 -953.747,E2 -953.747} C_VEL
LIN {X 0,Y 594.229,Z 601.956,A -85,B 0,C 180,E1 -954.694,E2 -954.694} C_VEL
LIN {X 0,Y 594.265,Z 598.533,A -85,B 0,C 180,E1 -955.879,E2 -955.879} C_VEL
LIN {X 0,Y 594.266,Z 593.502,A -85,B 0,C 180,E1 -957.106,E2 -957.106} C_VEL
LIN {X 0,Y 594.282,Z 587.984,A -85,B 0,C 180,E1 -958.136,E2 -958.136} C_VEL
LIN {X 0,Y 594.327,Z 580.537,A -85,B 0,C 180,E1 -959.24,E2 -959.24} C_VEL
LIN {X 0,Y 594.344,Z 572.245,A -85,B 0,C 180,E1 -960.221,E2 -960.221} C_VEL
LIN {X 0,Y 594.392,Z 563.8,A -85,B 0,C 180,E1 -961.041,E2 -961.041} C_VEL
LIN {X 0,Y 594.445,Z 553.385,A -85,B 0,C 180,E1 -961.871,E2 -961.871} C_VEL
LIN {X 0,Y 594.507,Z 542.83,A -85,B 0,C 180,E1 -962.545,E2 -962.545} C_VEL
LIN {X 0,Y 594.535,Z 530.468,A -85,B 0,C 180,E1 -963.165,E2 -963.165} C_VEL
LIN {X 0,Y 594.603,Z 518.454,A -85,B 0,C 180,E1 -963.618,E2 -963.618} C_VEL
LIN {X 0,Y 594.655,Z 505.312,A -85,B 0,C 180,E1 -963.964,E2 -963.964} C_VEL
LIN {X 0,Y 594.698,Z 489.509,A -85,B 0,C 180,E1 -964.2,E2 -964.2} C_VEL
LIN {X 0,Y 594.665,Z 396.016,A -85,B 0,C 180,E1 -965.334,E2 -965.334} C_VEL
LIN {X 0,Y 594.387,Z 394.084,A -85,B 0,C 180,E1 -965.381,E2 -965.381} C_VEL
LIN {X 0,Y 594.463,Z 377.583,A -85,B 0,C 180,E1 -968.135,E2 -968.135} C_VEL
LIN {X 0,Y 594.545,Z 359.87,A -85,B 0,C 180,E1 -971.134,E2 -971.134} C_VEL
LIN {X 0,Y 594.402,Z 357.442,A -85,B 0,C 180,E1 -971.561,E2 -971.561} C_VEL
LIN {X 0,Y 594.371,Z 357.446,A -85,B 0,C 180,E1 -974.218,E2 -974.218} C_VEL
LIN {X 0,Y 594.391,Z 357.445,A -85,B 0,C 180,E1 -976.32,E2 -976.32} C_VEL
LIN {X 0,Y 594.378,Z 357.443,A -85,B 0,C 180,E1 -979.094,E2 -979.094} C_VEL
LIN {X 0,Y 594.417,Z 357.437,A -85,B 0,C 180,E1 -981.843,E2 -981.843} C_VEL
LIN {X 0,Y 594.399,Z 357.446,A -85,B 0,C 180,E1 -984.571,E2 -984.571} C_VEL
LIN {X 0,Y 594.405,Z 357.437,A -85,B 0,C 180,E1 -987.288,E2 -987.288} C_VEL
LIN {X 0,Y 594.419,Z 357.44,A -85,B 0,C 180,E1 -989.999,E2 -989.999} C_VEL
LIN {X 0,Y 594.41,Z 357.44,A -85,B 0,C 180,E1 -992.71,E2 -992.71} C_VEL
LIN {X 0,Y 594.392,Z 357.439,A -85,B 0,C 180,E1 -995.427,E2 -995.427} C_VEL
LIN {X 0,Y 594.414,Z 357.447,A -85,B 0,C 180,E1 -998.156,E2 -998.156} C_VEL
LIN {X 0,Y 594.391,Z 357.439,A -85,B 0,C 180,E1 -1001.072,E2 -1001.072} C_VEL
LIN {X 0,Y 594.383,Z 357.444,A -85,B 0,C 180,E1 -1003.678,E2 -1003.678} C_VEL
LIN {X 0,Y 594.389,Z 357.44,A -85,B 0,C 180,E1 -1006.716,E2 -1006.716} C_VEL
LIN {X 0,Y 594.366,Z 357.444,A -85,B 0,C 180,E1 -1009.333,E2 -1009.333} C_VEL
LIN {X 0,Y 594.363,Z 357.446,A -85,B 0,C 180,E1 -1011.502,E2 -1011.502} C_VEL
LIN {X 0,Y 594.389,Z 357.441,A -85,B 0,C 180,E1 -1014.445,E2 -1014.445} C_VEL
LIN {X 0,Y 594.383,Z 357.44,A -85,B 0,C 180,E1 -1016.698,E2 -1016.698} C_VEL
LIN {X 0,Y 594.38,Z 357.441,A -85,B 0,C 180,E1 -1018.997,E2 -1018.997} C_VEL
LIN {X 0,Y 594.389,Z 357.448,A -85,B 0,C 180,E1 -1021.644,E2 -1021.644} C_VEL
LIN {X 0,Y 594.398,Z 357.438,A -85,B 0,C 180,E1 -1024.577,E2 -1024.577} C_VEL
LIN {X 0,Y 594.382,Z 357.443,A -85,B 0,C 180,E1 -1027.085,E2 -1027.085} C_VEL
LIN {X 0,Y 594.374,Z 357.448,A -85,B 0,C 180,E1 -1029.774,E2 -1029.774} C_VEL
LIN {X 0,Y 594.364,Z 357.443,A -85,B 0,C 180,E1 -1032.374,E2 -1032.374} C_VEL
LIN {X 0,Y 594.357,Z 357.449,A -85,B 0,C 180,E1 -1035.19,E2 -1035.19} C_VEL
LIN {X 0,Y 594.382,Z 357.449,A -85,B 0,C 180,E1 -1037.625,E2 -1037.625} C_VEL
LIN {X 0,Y 594.39,Z 357.449,A -85,B 0,C 180,E1 -1038.537,E2 -1038.537} C_VEL
LIN {X 0,Y 594.504,Z 369.244,A -85,B 0,C 180,E1 -1040.549,E2 -1040.549} C_VEL
LIN {X 0,Y 594.448,Z 386.851,A -85,B 0,C 180,E1 -1043.506,E2 -1043.506} C_VEL
LIN {X 0,Y 594.39,Z 394.362,A -85,B 0,C 180,E1 -1044.729,E2 -1044.729} C_VEL
LIN {X 0,Y 594.751,Z 399.984,A -85,B 0,C 180,E1 -1044.806,E2 -1044.806} C_VEL
LIN {X 0,Y 594.648,Z 501.383,A -85,B 0,C 180,E1 -1046.052,E2 -1046.052} C_VEL
LIN {X 0,Y 594.613,Z 515.032,A -85,B 0,C 180,E1 -1046.368,E2 -1046.368} C_VEL
LIN {X 0,Y 594.561,Z 527.714,A -85,B 0,C 180,E1 -1046.808,E2 -1046.808} C_VEL
LIN {X 0,Y 594.516,Z 539.448,A -85,B 0,C 180,E1 -1047.36,E2 -1047.36} C_VEL
LIN {X 0,Y 594.435,Z 551.152,A -85,B 0,C 180,E1 -1048.066,E2 -1048.066} C_VEL
LIN {X 0,Y 594.425,Z 561.53,A -85,B 0,C 180,E1 -1048.851,E2 -1048.851} C_VEL
LIN {X 0,Y 594.353,Z 570.378,A -85,B 0,C 180,E1 -1049.675,E2 -1049.675} C_VEL
LIN {X 0,Y 594.299,Z 578.62,A -85,B 0,C 180,E1 -1050.609,E2 -1050.609} C_VEL
LIN {X 0,Y 594.29,Z 585.703,A -85,B 0,C 180,E1 -1051.59,E2 -1051.59} C_VEL
LIN {X 0,Y 594.261,Z 591.239,A -85,B 0,C 180,E1 -1052.533,E2 -1052.533} C_VEL
LIN {X 0,Y 594.288,Z 596.535,A -85,B 0,C 180,E1 -1053.675,E2 -1053.675} C_VEL
LIN {X 0,Y 594.237,Z 600.404,A -85,B 0,C 180,E1 -1054.8,E2 -1054.8} C_VEL
LIN {X 0,Y 594.231,Z 602.384,A -85,B 0,C 180,E1 -1055.596,E2 -1055.596} C_VEL
LIN {X 0,Y 594.223,Z 603.646,A -85,B 0,C 180,E1 -1056.289,E2 -1056.289} C_VEL
LIN {X 0,Y 594.25,Z 604.728,A -85,B 0,C 180,E1 -1057.288,E2 -1057.288} C_VEL
LIN {X 0,Y 594.222,Z 604.905,A -85,B 0,C 180,E1 -1058.491,E2 -1058.491} C_VEL
LIN {X 0,Y 594.25,Z 604.396,A -85,B 0,C 180,E1 -1059.219,E2 -1059.219} C_VEL
LIN {X 0,Y 594.218,Z 603.42,A -85,B 0,C 180,E1 -1059.941,E2 -1059.941} C_VEL
LIN {X 0,Y 594.24,Z 600.884,A -85,B 0,C 180,E1 -1061.107,E2 -1061.107} C_VEL
LIN {X 0,Y 594.253,Z 597.751,A -85,B 0,C 180,E1 -1062.092,E2 -1062.092} C_VEL
LIN {X 0,Y 594.268,Z 592.496,A -85,B 0,C 180,E1 -1063.317,E2 -1063.317} C_VEL
LIN {X 0,Y 594.282,Z 586.41,A -85,B 0,C 180,E1 -1064.393,E2 -1064.393} C_VEL
LIN {X 0,Y 594.341,Z 578.89,A -85,B 0,C 180,E1 -1065.447,E2 -1065.447} C_VEL
LIN {X 0,Y 594.343,Z 571.283,A -85,B 0,C 180,E1 -1066.32,E2 -1066.32} C_VEL
LIN {X 0,Y 594.428,Z 562.072,A -85,B 0,C 180,E1 -1067.192,E2 -1067.192} C_VEL
LIN {X 0,Y 594.468,Z 551.9,A -85,B 0,C 180,E1 -1067.973,E2 -1067.973} C_VEL
LIN {X 0,Y 594.502,Z 540.755,A -85,B 0,C 180,E1 -1068.659,E2 -1068.659} C_VEL
LIN {X 0,Y 594.562,Z 528.971,A -85,B 0,C 180,E1 -1069.227,E2 -1069.227} C_VEL
LIN {X 0,Y 594.596,Z 517.186,A -85,B 0,C 180,E1 -1069.658,E2 -1069.658} C_VEL
LIN {X 0,Y 594.677,Z 504.316,A -85,B 0,C 180,E1 -1069.982,E2 -1069.982} C_VEL
LIN {X 0,Y 594.687,Z 486.159,A -85,B 0,C 180,E1 -1070.24,E2 -1070.24} C_VEL
LIN {X 0,Y 594.695,Z 395.995,A -85,B 0,C 180,E1 -1071.334,E2 -1071.334} C_VEL
LIN {X 0,Y 594.37,Z 394.143,A -85,B 0,C 180,E1 -1071.372,E2 -1071.372} C_VEL
LIN {X 0,Y 594.453,Z 378.019,A -85,B 0,C 180,E1 -1074.062,E2 -1074.062} C_VEL
LIN {X 0,Y 594.541,Z 362.933,A -85,B 0,C 180,E1 -1076.612,E2 -1076.612} C_VEL
LIN {X 0,Y 594.395,Z 357.443,A -85,B 0,C 180,E1 -1077.586,E2 -1077.586} C_VEL
LIN {X 0,Y 594.404,Z 357.44,A -85,B 0,C 180,E1 -1080,E2 -1080} C_VEL
LIN {X 0,Y 594.41,Z 357.445,A -85,B 0,C 180,E1 -1082.711,E2 -1082.711} C_VEL
LIN {X 0,Y 594.388,Z 357.44,A -85,B 0,C 180,E1 -1085.428,E2 -1085.428} C_VEL
LIN {X 0,Y 594.411,Z 357.444,A -85,B 0,C 180,E1 -1088.157,E2 -1088.157} C_VEL
LIN {X 0,Y 594.385,Z 357.441,A -85,B 0,C 180,E1 -1091.078,E2 -1091.078} C_VEL
LIN {X 0,Y 594.377,Z 357.444,A -85,B 0,C 180,E1 -1093.679,E2 -1093.679} C_VEL
LIN {X 0,Y 594.392,Z 357.441,A -85,B 0,C 180,E1 -1096.723,E2 -1096.723} C_VEL
LIN {X 0,Y 594.364,Z 357.444,A -85,B 0,C 180,E1 -1099.335,E2 -1099.335} C_VEL
LIN {X 0,Y 594.366,Z 357.446,A -85,B 0,C 180,E1 -1101.503,E2 -1101.503} C_VEL
LIN {X 0,Y 594.391,Z 357.447,A -85,B 0,C 180,E1 -1103.704,E2 -1103.704} C_VEL
LIN {X 0,Y 594.383,Z 357.441,A -85,B 0,C 180,E1 -1106.7,E2 -1106.7} C_VEL
LIN {X 0,Y 594.379,Z 357.442,A -85,B 0,C 180,E1 -1108.999,E2 -1108.999} C_VEL
LIN {X 0,Y 594.389,Z 357.45,A -85,B 0,C 180,E1 -1111.647,E2 -1111.647} C_VEL
LIN {X 0,Y 594.388,Z 357.44,A -85,B 0,C 180,E1 -1114.58,E2 -1114.58} C_VEL
LIN {X 0,Y 594.38,Z 357.445,A -85,B 0,C 180,E1 -1117.087,E2 -1117.087} C_VEL
LIN {X 0,Y 594.369,Z 357.446,A -85,B 0,C 180,E1 -1119.776,E2 -1119.776} C_VEL
LIN {X 0,Y 594.382,Z 357.441,A -85,B 0,C 180,E1 -1122.374,E2 -1122.374} C_VEL
LIN {X 0,Y 594.357,Z 357.453,A -85,B 0,C 180,E1 -1125.192,E2 -1125.192} C_VEL
LIN {X 0,Y 594.377,Z 357.441,A -85,B 0,C 180,E1 -1128.153,E2 -1128.153} C_VEL
LIN {X 0,Y 594.385,Z 357.448,A -85,B 0,C 180,E1 -1131.197,E2 -1131.197} C_VEL
LIN {X 0,Y 594.393,Z 357.44,A -85,B 0,C 180,E1 -1133.76,E2 -1133.76} C_VEL
LIN {X 0,Y 594.379,Z 357.442,A -85,B 0,C 180,E1 -1136.24,E2 -1136.24} C_VEL
LIN {X 0,Y 594.391,Z 357.447,A -85,B 0,C 180,E1 -1138.652,E2 -1138.652} C_VEL
LIN {X 0,Y 594.382,Z 357.446,A -85,B 0,C 180,E1 -1141.043,E2 -1141.043} C_VEL
LIN {X 0,Y 594.39,Z 357.441,A -85,B 0,C 180,E1 -1143.977,E2 -1143.977} C_VEL
LIN {X 0,Y 594.391,Z 357.446,A -85,B 0,C 180,E1 -1146.297,E2 -1146.297} C_VEL
LIN {X 0,Y 594.39,Z 357.531,A -85,B 0,C 180,E1 -1147.411,E2 -1147.411} C_VEL
LIN {X 0,Y 594.729,Z 362.51,A -85,B 0,C 180,E1 -1148.147,E2 -1148.147} C_VEL
LIN {X 0,Y 594.594,Z 382.517,A -85,B 0,C 180,E1 -1151.013,E2 -1151.013} C_VEL
LIN {X 0,Y 594.507,Z 401.549,A -85,B 0,C 180,E1 -1153.695,E2 -1153.695} C_VEL
LIN {X 0,Y 594.448,Z 422.8,A -85,B 0,C 180,E1 -1156.65,E2 -1156.65} C_VEL
LIN {X 0,Y 594.783,Z 426.803,A -85,B 0,C 180,E1 -1156.723,E2 -1156.723} C_VEL
LIN {X 0,Y 594.683,Z 531,A -85,B 0,C 180,E1 -1158,E2 -1158} C_VEL
LIN {X 0,Y 594.616,Z 544.253,A -85,B 0,C 180,E1 -1158.302,E2 -1158.302} C_VEL
LIN {X 0,Y 594.563,Z 556.43,A -85,B 0,C 180,E1 -1158.713,E2 -1158.713} C_VEL
LIN {X 0,Y 594.537,Z 568.651,A -85,B 0,C 180,E1 -1159.271,E2 -1159.271} C_VEL
LIN {X 0,Y 594.469,Z 580.215,A -85,B 0,C 180,E1 -1159.958,E2 -1159.958} C_VEL
LIN {X 0,Y 594.413,Z 590.608,A -85,B 0,C 180,E1 -1160.731,E2 -1160.731} C_VEL
LIN {X 0,Y 594.383,Z 599.122,A -85,B 0,C 180,E1 -1161.501,E2 -1161.501} C_VEL
LIN {X 0,Y 594.346,Z 606.968,A -85,B 0,C 180,E1 -1162.356,E2 -1162.356} C_VEL
LIN {X 0,Y 594.282,Z 614.817,A -85,B 0,C 180,E1 -1163.409,E2 -1163.409} C_VEL
LIN {X 0,Y 594.289,Z 621.685,A -85,B 0,C 180,E1 -1164.572,E2 -1164.572} C_VEL
LIN {X 0,Y 594.27,Z 626.375,A -85,B 0,C 180,E1 -1165.592,E2 -1165.592} C_VEL
LIN {X 0,Y 594.267,Z 629.959,A -85,B 0,C 180,E1 -1166.611,E2 -1166.611} C_VEL
LIN {X 0,Y 594.226,Z 631.811,A -85,B 0,C 180,E1 -1167.289,E2 -1167.289} C_VEL
LIN {X 0,Y 594.24,Z 633.203,A -85,B 0,C 180,E1 -1167.968,E2 -1167.968} C_VEL
LIN {X 0,Y 594.239,Z 634.785,A -85,B 0,C 180,E1 -1169.323,E2 -1169.323} C_VEL
LIN {X 0,Y 594.236,Z 635,A -85,B 0,C 180,E1 -1170.001,E2 -1170.001} C_VEL
LIN {X 0,Y 594.247,Z 634.184,A -85,B 0,C 180,E1 -1171.356,E2 -1171.356} C_VEL
LIN {X 0,Y 594.24,Z 633.2,A -85,B 0,C 180,E1 -1172.034,E2 -1172.034} C_VEL
LIN {X 0,Y 594.226,Z 631.807,A -85,B 0,C 180,E1 -1172.712,E2 -1172.712} C_VEL
LIN {X 0,Y 594.289,Z 628.893,A -85,B 0,C 180,E1 -1173.73,E2 -1173.73} C_VEL
LIN {X 0,Y 594.242,Z 624.946,A -85,B 0,C 180,E1 -1174.75,E2 -1174.75} C_VEL
LIN {X 0,Y 594.304,Z 618.872,A -85,B 0,C 180,E1 -1175.94,E2 -1175.94} C_VEL
LIN {X 0,Y 594.309,Z 612.23,A -85,B 0,C 180,E1 -1176.963,E2 -1176.963} C_VEL
LIN {X 0,Y 594.359,Z 603.983,A -85,B 0,C 180,E1 -1177.987,E2 -1177.987} C_VEL
LIN {X 0,Y 594.382,Z 595.528,A -85,B 0,C 180,E1 -1178.843,E2 -1178.843} C_VEL
LIN {X 0,Y 594.422,Z 585.083,A -85,B 0,C 180,E1 -1179.7,E2 -1179.7} C_VEL
LIN {X 0,Y 594.482,Z 574.746,A -85,B 0,C 180,E1 -1180.387,E2 -1180.387} C_VEL
LIN {X 0,Y 594.56,Z 563.704,A -85,B 0,C 180,E1 -1180.974,E2 -1180.974} C_VEL
LIN {X 0,Y 594.583,Z 551.686,A -85,B 0,C 180,E1 -1181.465,E2 -1181.465} C_VEL
LIN {X 0,Y 594.637,Z 538.317,A -85,B 0,C 180,E1 -1181.851,E2 -1181.851} C_VEL
LIN {X 0,Y 594.693,Z 525.024,A -85,B 0,C 180,E1 -1182.088,E2 -1182.088} C_VEL
LIN {X 0,Y 594.63,Z 424.196,A -85,B 0,C 180,E1 -1183.312,E2 -1183.312} C_VEL
LIN {X 0,Y 594.448,Z 422.787,A -85,B 0,C 180,E1 -1183.352,E2 -1183.352} C_VEL
LIN {X 0,Y 594.509,Z 401.536,A -85,B 0,C 180,E1 -1186.306,E2 -1186.306} C_VEL
LIN {X 0,Y 594.631,Z 381.719,A -85,B 0,C 180,E1 -1189.1,E2 -1189.1} C_VEL
LIN {X 0,Y 594.731,Z 362.497,A -85,B 0,C 180,E1 -1191.855,E2 -1191.855} C_VEL
LIN {X 0,Y 594.395,Z 357.445,A -85,B 0,C 180,E1 -1192.625,E2 -1192.625} C_VEL
LIN {X 0,Y 594.382,Z 357.448,A -85,B 0,C 180,E1 -1195.194,E2 -1195.194} C_VEL
LIN {X 0,Y 594.392,Z 357.447,A -85,B 0,C 180,E1 -1197.527,E2 -1197.527} C_VEL
LIN {X 0,Y 594.393,Z 357.439,A -85,B 0,C 180,E1 -1200.329,E2 -1200.329} C_VEL
LIN {X 0,Y 594.383,Z 357.446,A -85,B 0,C 180,E1 -1202.951,E2 -1202.951} C_VEL
LIN {X 0,Y 594.362,Z 357.45,A -85,B 0,C 180,E1 -1205.409,E2 -1205.409} C_VEL
LIN {X 0,Y 594.389,Z 357.44,A -85,B 0,C 180,E1 -1207.941,E2 -1207.941} C_VEL
LIN {X 0,Y 594.38,Z 357.447,A -85,B 0,C 180,E1 -1210.822,E2 -1210.822} C_VEL
LIN {X 0,Y 594.373,Z 357.442,A -85,B 0,C 180,E1 -1213.84,E2 -1213.84} C_VEL
LIN {X 0,Y 594.372,Z 357.448,A -85,B 0,C 180,E1 -1216.701,E2 -1216.701} C_VEL
LIN {X 0,Y 594.371,Z 357.444,A -85,B 0,C 180,E1 -1219.433,E2 -1219.433} C_VEL
LIN {X 0,Y 594.394,Z 357.442,A -85,B 0,C 180,E1 -1222.392,E2 -1222.392} C_VEL
LIN {X 0,Y 594.381,Z 357.442,A -85,B 0,C 180,E1 -1225.42,E2 -1225.42} C_VEL
LIN {X 0,Y 594.381,Z 357.445,A -85,B 0,C 180,E1 -1228.358,E2 -1228.358} C_VEL
LIN {X 0,Y 594.387,Z 357.444,A -85,B 0,C 180,E1 -1231.042,E2 -1231.042} C_VEL
LIN {X 0,Y 594.387,Z 357.441,A -85,B 0,C 180,E1 -1233.978,E2 -1233.978} C_VEL
LIN {X 0,Y 594.388,Z 357.446,A -85,B 0,C 180,E1 -1236.296,E2 -1236.296} C_VEL
LIN {X 0,Y 594.405,Z 357.438,A -85,B 0,C 180,E1 -1239.224,E2 -1239.224} C_VEL
LIN {X 0,Y 594.35,Z 357.448,A -85,B 0,C 180,E1 -1242.095,E2 -1242.095} C_VEL
LIN {X 0,Y 594.367,Z 357.45,A -85,B 0,C 180,E1 -1244.219,E2 -1244.219} C_VEL
LIN {X 0,Y 594.381,Z 357.45,A -85,B 0,C 180,E1 -1246.321,E2 -1246.321} C_VEL
LIN {X 0,Y 594.378,Z 357.441,A -85,B 0,C 180,E1 -1249.095,E2 -1249.095} C_VEL
LIN {X 0,Y 594.418,Z 357.44,A -85,B 0,C 180,E1 -1251.843,E2 -1251.843} C_VEL
LIN {X 0,Y 594.394,Z 357.443,A -85,B 0,C 180,E1 -1254.572,E2 -1254.572} C_VEL
LIN {X 0,Y 594.412,Z 357.436,A -85,B 0,C 180,E1 -1257.289,E2 -1257.289} C_VEL
LIN {X 0,Y 594.419,Z 357.445,A -85,B 0,C 180,E1 -1260,E2 -1260} C_VEL
LIN {X 0,Y 594.412,Z 357.438,A -85,B 0,C 180,E1 -1262.711,E2 -1262.711} C_VEL
LIN {X 0,Y 594.395,Z 357.441,A -85,B 0,C 180,E1 -1265.428,E2 -1265.428} C_VEL
LIN {X 0,Y 594.419,Z 357.442,A -85,B 0,C 180,E1 -1268.157,E2 -1268.157} C_VEL
LIN {X 0,Y 594.393,Z 357.44,A -85,B 0,C 180,E1 -1271.073,E2 -1271.073} C_VEL
LIN {X 0,Y 594.386,Z 357.448,A -85,B 0,C 180,E1 -1273.679,E2 -1273.679} C_VEL
LIN {X 0,Y 594.365,Z 357.446,A -85,B 0,C 180,E1 -1275.326,E2 -1275.326} C_VEL
LIN {X 0,Y 593.692,Z 357.536,A -85,B 0,C 180,E1 -1275.892,E2 -1275.892} C_VEL
LIN {X 0,Y 590.825,Z 357.894,A -85,B 0,C 180,E1 -1276.81,E2 -1276.81} C_VEL
LIN {X 0,Y 588.414,Z 358.192,A -85,B 0,C 180,E1 -1277.548,E2 -1277.548} C_VEL
LIN {X 0,Y 587.39,Z 358.316,A -85,B 0,C 180,E1 -1278.118,E2 -1278.118} C_VEL
LIN {X 0,Y 587.313,Z 358.323,A -85,B 0,C 180,E1 -1278.311,E2 -1278.311} C_VEL
LIN {X 0,Y 587.337,Z 358.32,A -85,B 0,C 180,E1 -1281.038,E2 -1281.038} C_VEL
LIN {X 0,Y 587.326,Z 358.324,A -85,B 0,C 180,E1 -1283.259,E2 -1283.259} C_VEL
LIN {X 0,Y 587.34,Z 358.328,A -85,B 0,C 180,E1 -1285.517,E2 -1285.517} C_VEL
LIN {X 0,Y 587.345,Z 358.323,A -85,B 0,C 180,E1 -1287.818,E2 -1287.818} C_VEL
LIN {X 0,Y 587.341,Z 358.319,A -85,B 0,C 180,E1 -1290.509,E2 -1290.509} C_VEL
LIN {X 0,Y 587.379,Z 358.493,A -85,B 0,C 180,E1 -1292.475,E2 -1292.475} C_VEL
LIN {X 0,Y 587.483,Z 369.435,A -85,B 0,C 180,E1 -1294.366,E2 -1294.366} C_VEL
LIN {X 0,Y 587.405,Z 385.927,A -85,B 0,C 180,E1 -1297.172,E2 -1297.172} C_VEL
LIN {X 0,Y 587.358,Z 394.233,A -85,B 0,C 180,E1 -1298.565,E2 -1298.565} C_VEL
LIN {X 0,Y 587.869,Z 398.611,A -85,B 0,C 180,E1 -1298.631,E2 -1298.631} C_VEL
LIN {X 0,Y 587.726,Z 501.517,A -85,B 0,C 180,E1 -1299.911,E2 -1299.911} C_VEL
LIN {X 0,Y 587.664,Z 514.957,A -85,B 0,C 180,E1 -1300.226,E2 -1300.226} C_VEL
LIN {X 0,Y 587.609,Z 527.886,A -85,B 0,C 180,E1 -1300.681,E2 -1300.681} C_VEL
LIN {X 0,Y 587.549,Z 539.863,A -85,B 0,C 180,E1 -1301.253,E2 -1301.253} C_VEL
LIN {X 0,Y 587.486,Z 551.15,A -85,B 0,C 180,E1 -1301.946,E2 -1301.946} C_VEL
LIN {X 0,Y 587.351,Z 561.875,A -85,B 0,C 180,E1 -1302.769,E2 -1302.769} C_VEL
LIN {X 0,Y 587.308,Z 571.873,A -85,B 0,C 180,E1 -1303.73,E2 -1303.73} C_VEL
LIN {X 0,Y 587.263,Z 580.487,A -85,B 0,C 180,E1 -1304.757,E2 -1304.757} C_VEL
LIN {X 0,Y 587.222,Z 588.086,A -85,B 0,C 180,E1 -1305.898,E2 -1305.898} C_VEL
LIN {X 0,Y 587.198,Z 593.78,A -85,B 0,C 180,E1 -1306.982,E2 -1306.982} C_VEL
LIN {X 0,Y 587.17,Z 597.623,A -85,B 0,C 180,E1 -1307.911,E2 -1307.911} C_VEL
LIN {X 0,Y 587.137,Z 600.904,A -85,B 0,C 180,E1 -1308.948,E2 -1308.948} C_VEL
LIN {X 0,Y 587.139,Z 603.227,A -85,B 0,C 180,E1 -1310.003,E2 -1310.003} C_VEL
LIN {X 0,Y 587.113,Z 604.598,A -85,B 0,C 180,E1 -1311.085,E2 -1311.085} C_VEL
LIN {X 0,Y 587.143,Z 604.931,A -85,B 0,C 180,E1 -1312.376,E2 -1312.376} C_VEL
LIN {X 0,Y 587.128,Z 604.292,A -85,B 0,C 180,E1 -1313.322,E2 -1313.322} C_VEL
LIN {X 0,Y 587.139,Z 602.46,A -85,B 0,C 180,E1 -1314.484,E2 -1314.484} C_VEL
LIN {X 0,Y 587.162,Z 599.067,A -85,B 0,C 180,E1 -1315.766,E2 -1315.766} C_VEL
LIN {X 0,Y 587.169,Z 594.673,A -85,B 0,C 180,E1 -1316.914,E2 -1316.914} C_VEL
LIN {X 0,Y 587.215,Z 589.087,A -85,B 0,C 180,E1 -1318.021,E2 -1318.021} C_VEL
LIN {X 0,Y 587.253,Z 582.695,A -85,B 0,C 180,E1 -1319.028,E2 -1319.028} C_VEL
LIN {X 0,Y 587.291,Z 574.889,A -85,B 0,C 180,E1 -1320.025,E2 -1320.025} C_VEL
LIN {X 0,Y 587.358,Z 566.173,A -85,B 0,C 180,E1 -1320.934,E2 -1320.934} C_VEL
LIN {X 0,Y 587.408,Z 555.973,A -85,B 0,C 180,E1 -1321.796,E2 -1321.796} C_VEL
LIN {X 0,Y 587.511,Z 544.437,A -85,B 0,C 180,E1 -1322.577,E2 -1322.577} C_VEL
LIN {X 0,Y 587.568,Z 532.559,A -85,B 0,C 180,E1 -1323.205,E2 -1323.205} C_VEL
LIN {X 0,Y 587.643,Z 520.521,A -85,B 0,C 180,E1 -1323.688,E2 -1323.688} C_VEL
LIN {X 0,Y 587.701,Z 506.896,A -85,B 0,C 180,E1 -1324.072,E2 -1324.072} C_VEL
LIN {X 0,Y 587.749,Z 493.216,A -85,B 0,C 180,E1 -1324.3,E2 -1324.3} C_VEL
LIN {X 0,Y 587.793,Z 396.864,A -85,B 0,C 180,E1 -1325.482,E2 -1325.482} C_VEL
LIN {X 0,Y 587.355,Z 394.1,A -85,B 0,C 180,E1 -1325.541,E2 -1325.541} C_VEL
LIN {X 0,Y 587.462,Z 377.097,A -85,B 0,C 180,E1 -1328.415,E2 -1328.415} C_VEL
LIN {X 0,Y 587.553,Z 360.054,A -85,B 0,C 180,E1 -1331.338,E2 -1331.338} C_VEL
LIN {X 0,Y 587.374,Z 358.318,A -85,B 0,C 180,E1 -1331.649,E2 -1331.649} C_VEL
LIN {X 0,Y 587.328,Z 358.322,A -85,B 0,C 180,E1 -1334.024,E2 -1334.024} C_VEL
LIN {X 0,Y 587.367,Z 358.318,A -85,B 0,C 180,E1 -1336.154,E2 -1336.154} C_VEL
LIN {X 0,Y 587.345,Z 358.321,A -85,B 0,C 180,E1 -1338.962,E2 -1338.962} C_VEL
LIN {X 0,Y 587.369,Z 358.314,A -85,B 0,C 180,E1 -1341.744,E2 -1341.744} C_VEL
LIN {X 0,Y 587.363,Z 358.324,A -85,B 0,C 180,E1 -1344.506,E2 -1344.506} C_VEL
LIN {X 0,Y 587.372,Z 358.314,A -85,B 0,C 180,E1 -1347.256,E2 -1347.256} C_VEL
LIN {X 0,Y 587.388,Z 358.316,A -85,B 0,C 180,E1 -1349.999,E2 -1349.999} C_VEL
LIN {X 0,Y 587.376,Z 358.316,A -85,B 0,C 180,E1 -1352.742,E2 -1352.742} C_VEL
LIN {X 0,Y 587.358,Z 358.316,A -85,B 0,C 180,E1 -1355.492,E2 -1355.492} C_VEL
LIN {X 0,Y 587.366,Z 358.323,A -85,B 0,C 180,E1 -1358.254,E2 -1358.254} C_VEL
LIN {X 0,Y 587.351,Z 358.316,A -85,B 0,C 180,E1 -1361.133,E2 -1361.133} C_VEL
LIN {X 0,Y 587.368,Z 358.321,A -85,B 0,C 180,E1 -1364.259,E2 -1364.259} C_VEL
LIN {X 0,Y 587.355,Z 358.317,A -85,B 0,C 180,E1 -1367.405,E2 -1367.405} C_VEL
LIN {X 0,Y 587.327,Z 358.323,A -85,B 0,C 180,E1 -1370.304,E2 -1370.304} C_VEL
LIN {X 0,Y 587.322,Z 358.321,A -85,B 0,C 180,E1 -1373.258,E2 -1373.258} C_VEL
LIN {X 0,Y 587.334,Z 358.323,A -85,B 0,C 180,E1 -1375.515,E2 -1375.515} C_VEL
LIN {X 0,Y 587.347,Z 358.327,A -85,B 0,C 180,E1 -1377.816,E2 -1377.816} C_VEL
LIN {X 0,Y 587.349,Z 358.317,A -85,B 0,C 180,E1 -1380.511,E2 -1380.511} C_VEL
LIN {X 0,Y 587.333,Z 358.324,A -85,B 0,C 180,E1 -1383.395,E2 -1383.395} C_VEL
LIN {X 0,Y 587.355,Z 358.322,A -85,B 0,C 180,E1 -1385.894,E2 -1385.894} C_VEL
LIN {X 0,Y 587.329,Z 358.319,A -85,B 0,C 180,E1 -1388.478,E2 -1388.478} C_VEL
LIN {X 0,Y 587.334,Z 358.322,A -85,B 0,C 180,E1 -1391.155,E2 -1391.155} C_VEL
LIN {X 0,Y 587.329,Z 358.321,A -85,B 0,C 180,E1 -1394.113,E2 -1394.113} C_VEL
LIN {X 0,Y 587.332,Z 358.323,A -85,B 0,C 180,E1 -1396.995,E2 -1396.995} C_VEL
LIN {X 0,Y 587.394,Z 358.398,A -85,B 0,C 180,E1 -1398.459,E2 -1398.459} C_VEL
LIN {X 0,Y 587.512,Z 368.074,A -85,B 0,C 180,E1 -1400.133,E2 -1400.133} C_VEL
LIN {X 0,Y 587.418,Z 385.166,A -85,B 0,C 180,E1 -1403.044,E2 -1403.044} C_VEL
LIN {X 0,Y 587.354,Z 394.208,A -85,B 0,C 180,E1 -1404.565,E2 -1404.565} C_VEL
LIN {X 0,Y 587.859,Z 398.506,A -85,B 0,C 180,E1 -1404.63,E2 -1404.63} C_VEL
LIN {X 0,Y 587.711,Z 501.192,A -85,B 0,C 180,E1 -1405.906,E2 -1405.906} C_VEL
LIN {X 0,Y 587.681,Z 514.547,A -85,B 0,C 180,E1 -1406.214,E2 -1406.214} C_VEL
LIN {X 0,Y 587.594,Z 526.4,A -85,B 0,C 180,E1 -1406.62,E2 -1406.62} C_VEL
LIN {X 0,Y 587.54,Z 538.009,A -85,B 0,C 180,E1 -1407.155,E2 -1407.155} C_VEL
LIN {X 0,Y 587.459,Z 549.342,A -85,B 0,C 180,E1 -1407.824,E2 -1407.824} C_VEL
LIN {X 0,Y 587.373,Z 560.27,A -85,B 0,C 180,E1 -1408.635,E2 -1408.635} C_VEL
LIN {X 0,Y 587.345,Z 569.544,A -85,B 0,C 180,E1 -1409.486,E2 -1409.486} C_VEL
LIN {X 0,Y 587.253,Z 577.817,A -85,B 0,C 180,E1 -1410.418,E2 -1410.418} C_VEL
LIN {X 0,Y 587.222,Z 584.957,A -85,B 0,C 180,E1 -1411.397,E2 -1411.397} C_VEL
LIN {X 0,Y 587.196,Z 590.537,A -85,B 0,C 180,E1 -1412.333,E2 -1412.333} C_VEL
LIN {X 0,Y 587.196,Z 595.337,A -85,B 0,C 180,E1 -1413.331,E2 -1413.331} C_VEL
LIN {X 0,Y 587.143,Z 599.535,A -85,B 0,C 180,E1 -1414.474,E2 -1414.474} C_VEL
LIN {X 0,Y 587.131,Z 602.173,A -85,B 0,C 180,E1 -1415.464,E2 -1415.464} C_VEL
LIN {X 0,Y 587.117,Z 604.256,A -85,B 0,C 180,E1 -1416.732,E2 -1416.732} C_VEL
LIN {X 0,Y 587.147,Z 604.862,A -85,B 0,C 180,E1 -1417.478,E2 -1417.478} C_VEL
LIN {X 0,Y 587.138,Z 604.969,A -85,B 0,C 180,E1 -1418.218,E2 -1418.218} C_VEL
LIN {X 0,Y 587.163,Z 604.59,A -85,B 0,C 180,E1 -1419.002,E2 -1419.002} C_VEL
LIN {X 0,Y 587.148,Z 603.858,A -85,B 0,C 180,E1 -1419.688,E2 -1419.688} C_VEL
LIN {X 0,Y 587.148,Z 601.221,A -85,B 0,C 180,E1 -1421.011,E2 -1421.011} C_VEL
LIN {X 0,Y 587.172,Z 597.432,A -85,B 0,C 180,E1 -1422.229,E2 -1422.229} C_VEL
LIN {X 0,Y 587.175,Z 592.847,A -85,B 0,C 180,E1 -1423.306,E2 -1423.306} C_VEL
LIN {X 0,Y 587.198,Z 586.995,A -85,B 0,C 180,E1 -1424.377,E2 -1424.377} C_VEL
LIN {X 0,Y 587.279,Z 579.601,A -85,B 0,C 180,E1 -1425.445,E2 -1425.445} C_VEL
LIN {X 0,Y 587.295,Z 572.128,A -85,B 0,C 180,E1 -1426.329,E2 -1426.329} C_VEL
LIN {X 0,Y 587.38,Z 563.087,A -85,B 0,C 180,E1 -1427.211,E2 -1427.211} C_VEL
LIN {X 0,Y 587.432,Z 553.202,A -85,B 0,C 180,E1 -1428.002,E2 -1428.002} C_VEL
LIN {X 0,Y 587.505,Z 542.159,A -85,B 0,C 180,E1 -1428.708,E2 -1428.708} C_VEL
LIN {X 0,Y 587.585,Z 530.007,A -85,B 0,C 180,E1 -1429.316,E2 -1429.316} C_VEL
LIN {X 0,Y 587.643,Z 518.516,A -85,B 0,C 180,E1 -1429.752,E2 -1429.752} C_VEL
LIN {X 0,Y 587.722,Z 505.558,A -85,B 0,C 180,E1 -1430.102,E2 -1430.102} C_VEL
LIN {X 0,Y 587.782,Z 489.759,A -85,B 0,C 180,E1 -1430.342,E2 -1430.342} C_VEL
LIN {X 0,Y 587.802,Z 396.981,A -85,B 0,C 180,E1 -1431.48,E2 -1431.48} C_VEL
LIN {X 0,Y 587.352,Z 394.179,A -85,B 0,C 180,E1 -1431.528,E2 -1431.528} C_VEL
LIN {X 0,Y 587.428,Z 377.57,A -85,B 0,C 180,E1 -1434.335,E2 -1434.335} C_VEL
LIN {X 0,Y 587.523,Z 362.512,A -85,B 0,C 180,E1 -1436.914,E2 -1436.914} C_VEL
LIN {X 0,Y 587.35,Z 358.321,A -85,B 0,C 180,E1 -1437.685,E2 -1437.685} C_VEL
LIN {X 0,Y 587.373,Z 358.316,A -85,B 0,C 180,E1 -1440,E2 -1440} C_VEL
LIN {X 0,Y 587.375,Z 358.321,A -85,B 0,C 180,E1 -1442.743,E2 -1442.743} C_VEL
LIN {X 0,Y 587.353,Z 358.317,A -85,B 0,C 180,E1 -1445.493,E2 -1445.493} C_VEL
LIN {X 0,Y 587.364,Z 358.324,A -85,B 0,C 180,E1 -1448.255,E2 -1448.255} C_VEL
LIN {X 0,Y 587.351,Z 358.317,A -85,B 0,C 180,E1 -1451.142,E2 -1451.142} C_VEL
LIN {X 0,Y 587.355,Z 358.325,A -85,B 0,C 180,E1 -1454.261,E2 -1454.261} C_VEL
LIN {X 0,Y 587.354,Z 358.317,A -85,B 0,C 180,E1 -1457.406,E2 -1457.406} C_VEL
LIN {X 0,Y 587.328,Z 358.324,A -85,B 0,C 180,E1 -1460.305,E2 -1460.305} C_VEL
LIN {X 0,Y 587.361,Z 358.317,A -85,B 0,C 180,E1 -1463.257,E2 -1463.257} C_VEL
LIN {X 0,Y 587.358,Z 358.319,A -85,B 0,C 180,E1 -1466.278,E2 -1466.278} C_VEL
LIN {X 0,Y 587.347,Z 358.319,A -85,B 0,C 180,E1 -1469.135,E2 -1469.135} C_VEL
LIN {X 0,Y 587.352,Z 358.323,A -85,B 0,C 180,E1 -1471.839,E2 -1471.839} C_VEL
LIN {X 0,Y 587.35,Z 358.317,A -85,B 0,C 180,E1 -1474.35,E2 -1474.35} C_VEL
LIN {X 0,Y 587.345,Z 358.318,A -85,B 0,C 180,E1 -1476.747,E2 -1476.747} C_VEL
LIN {X 0,Y 587.339,Z 358.328,A -85,B 0,C 180,E1 -1479.36,E2 -1479.36} C_VEL
LIN {X 0,Y 587.331,Z 358.319,A -85,B 0,C 180,E1 -1482.109,E2 -1482.109} C_VEL
LIN {X 0,Y 587.31,Z 358.329,A -85,B 0,C 180,E1 -1485.09,E2 -1485.09} C_VEL
LIN {X 0,Y 587.347,Z 358.318,A -85,B 0,C 180,E1 -1487.929,E2 -1487.929} C_VEL
LIN {X 0,Y 587.333,Z 358.329,A -85,B 0,C 180,E1 -1491.059,E2 -1491.059} C_VEL
LIN {X 0,Y 587.351,Z 358.322,A -85,B 0,C 180,E1 -1493.292,E2 -1493.292} C_VEL
LIN {X 0,Y 587.366,Z 358.315,A -85,B 0,C 180,E1 -1495.782,E2 -1495.782} C_VEL
LIN {X 0,Y 587.35,Z 358.318,A -85,B 0,C 180,E1 -1498.233,E2 -1498.233} C_VEL
LIN {X 0,Y 587.35,Z 358.325,A -85,B 0,C 180,E1 -1500.867,E2 -1500.867} C_VEL
LIN {X 0,Y 587.361,Z 358.316,A -85,B 0,C 180,E1 -1503.819,E2 -1503.819} C_VEL
LIN {X 0,Y 587.337,Z 358.321,A -85,B 0,C 180,E1 -1505.995,E2 -1505.995} C_VEL
LIN {X 0,Y 587.344,Z 358.447,A -85,B 0,C 180,E1 -1507.26,E2 -1507.26} C_VEL
LIN {X 0,Y 587.822,Z 362.51,A -85,B 0,C 180,E1 -1507.877,E2 -1507.877} C_VEL
LIN {X 0,Y 587.671,Z 383.132,A -85,B 0,C 180,E1 -1510.869,E2 -1510.869} C_VEL
LIN {X 0,Y 587.53,Z 402.808,A -85,B 0,C 180,E1 -1513.675,E2 -1513.675} C_VEL
LIN {X 0,Y 587.387,Z 422.8,A -85,B 0,C 180,E1 -1516.487,E2 -1516.487} C_VEL
LIN {X 0,Y 587.884,Z 426.803,A -85,B 0,C 180,E1 -1516.564,E2 -1516.564} C_VEL
LIN {X 0,Y 587.747,Z 530.999,A -85,B 0,C 180,E1 -1517.857,E2 -1517.857} C_VEL
LIN {X 0,Y 587.667,Z 544.254,A -85,B 0,C 180,E1 -1518.161,E2 -1518.161} C_VEL
LIN {X 0,Y 587.589,Z 556.62,A -85,B 0,C 180,E1 -1518.584,E2 -1518.584} C_VEL
LIN {X 0,Y 587.552,Z 568.649,A -85,B 0,C 180,E1 -1519.142,E2 -1519.142} C_VEL
LIN {X 0,Y 587.465,Z 580.216,A -85,B 0,C 180,E1 -1519.837,E2 -1519.837} C_VEL
LIN {X 0,Y 587.391,Z 590.61,A -85,B 0,C 180,E1 -1520.619,E2 -1520.619} C_VEL
LIN {X 0,Y 587.321,Z 599.122,A -85,B 0,C 180,E1 -1521.399,E2 -1521.399} C_VEL
LIN {X 0,Y 587.273,Z 606.969,A -85,B 0,C 180,E1 -1522.264,E2 -1522.264} C_VEL
LIN {X 0,Y 587.231,Z 613.476,A -85,B 0,C 180,E1 -1523.127,E2 -1523.127} C_VEL
LIN {X 0,Y 587.236,Z 619.872,A -85,B 0,C 180,E1 -1524.162,E2 -1524.162} C_VEL
LIN {X 0,Y 587.147,Z 624.954,A -85,B 0,C 180,E1 -1525.195,E2 -1525.195} C_VEL
LIN {X 0,Y 587.212,Z 628.899,A -85,B 0,C 180,E1 -1526.227,E2 -1526.227} C_VEL
LIN {X 0,Y 587.132,Z 631.811,A -85,B 0,C 180,E1 -1527.257,E2 -1527.257} C_VEL
LIN {X 0,Y 587.139,Z 633.202,A -85,B 0,C 180,E1 -1527.943,E2 -1527.943} C_VEL
LIN {X 0,Y 587.14,Z 634.785,A -85,B 0,C 180,E1 -1529.315,E2 -1529.315} C_VEL
LIN {X 0,Y 587.137,Z 635,A -85,B 0,C 180,E1 -1530.001,E2 -1530.001} C_VEL
LIN {X 0,Y 587.147,Z 634.184,A -85,B 0,C 180,E1 -1531.373,E2 -1531.373} C_VEL
LIN {X 0,Y 587.139,Z 633.2,A -85,B 0,C 180,E1 -1532.059,E2 -1532.059} C_VEL
LIN {X 0,Y 587.132,Z 631.808,A -85,B 0,C 180,E1 -1532.745,E2 -1532.745} C_VEL
LIN {X 0,Y 587.212,Z 628.893,A -85,B 0,C 180,E1 -1533.775,E2 -1533.775} C_VEL
LIN {X 0,Y 587.147,Z 624.946,A -85,B 0,C 180,E1 -1534.807,E2 -1534.807} C_VEL
LIN {X 0,Y 587.217,Z 618.872,A -85,B 0,C 180,E1 -1536.012,E2 -1536.012} C_VEL
LIN {X 0,Y 587.246,Z 612.231,A -85,B 0,C 180,E1 -1537.047,E2 -1537.047} C_VEL
LIN {X 0,Y 587.3,Z 603.983,A -85,B 0,C 180,E1 -1538.084,E2 -1538.084} C_VEL
LIN {X 0,Y 587.344,Z 595.529,A -85,B 0,C 180,E1 -1538.95,E2 -1538.95} C_VEL
LIN {X 0,Y 587.414,Z 585.084,A -85,B 0,C 180,E1 -1539.817,E2 -1539.817} C_VEL
LIN {X 0,Y 587.496,Z 574.744,A -85,B 0,C 180,E1 -1540.512,E2 -1540.512} C_VEL
LIN {X 0,Y 587.585,Z 562.793,A -85,B 0,C 180,E1 -1541.149,E2 -1541.149} C_VEL
LIN {X 0,Y 587.628,Z 550.572,A -85,B 0,C 180,E1 -1541.64,E2 -1541.64} C_VEL
LIN {X 0,Y 587.711,Z 537.402,A -85,B 0,C 180,E1 -1542.015,E2 -1542.015} C_VEL
LIN {X 0,Y 587.775,Z 525.024,A -85,B 0,C 180,E1 -1542.232,E2 -1542.232} C_VEL
LIN {X 0,Y 587.711,Z 424.764,A -85,B 0,C 180,E1 -1543.465,E2 -1543.465} C_VEL
LIN {X 0,Y 587.387,Z 422.787,A -85,B 0,C 180,E1 -1543.515,E2 -1543.515} C_VEL
LIN {X 0,Y 587.532,Z 402.795,A -85,B 0,C 180,E1 -1546.327,E2 -1546.327} C_VEL
LIN {X 0,Y 587.673,Z 383.128,A -85,B 0,C 180,E1 -1549.132,E2 -1549.132} C_VEL
LIN {X 0,Y 587.824,Z 362.497,A -85,B 0,C 180,E1 -1552.125,E2 -1552.125} C_VEL
LIN {X 0,Y 587.337,Z 358.325,A -85,B 0,C 180,E1 -1552.792,E2 -1552.792} C_VEL
LIN {X 0,Y 587.341,Z 358.327,A -85,B 0,C 180,E1 -1555.517,E2 -1555.517} C_VEL
LIN {X 0,Y 587.352,Z 358.32,A -85,B 0,C 180,E1 -1557.818,E2 -1557.818} C_VEL
LIN {X 0,Y 587.348,Z 358.318,A -85,B 0,C 180,E1 -1560.511,E2 -1560.511} C_VEL
LIN {X 0,Y 587.34,Z 358.325,A -85,B 0,C 180,E1 -1563.397,E2 -1563.397} C_VEL
LIN {X 0,Y 587.299,Z 358.324,A -85,B 0,C 180,E1 -1565.9,E2 -1565.9} C_VEL
LIN {X 0,Y 587.337,Z 358.32,A -85,B 0,C 180,E1 -1568.48,E2 -1568.48} C_VEL
LIN {X 0,Y 587.34,Z 358.327,A -85,B 0,C 180,E1 -1571.157,E2 -1571.157} C_VEL
LIN {X 0,Y 587.332,Z 358.319,A -85,B 0,C 180,E1 -1574.114,E2 -1574.114} C_VEL
LIN {X 0,Y 587.32,Z 358.33,A -85,B 0,C 180,E1 -1576.994,E2 -1576.994} C_VEL
LIN {X 0,Y 587.316,Z 358.321,A -85,B 0,C 180,E1 -1579.746,E2 -1579.746} C_VEL
LIN {X 0,Y 587.349,Z 358.32,A -85,B 0,C 180,E1 -1582.392,E2 -1582.392} C_VEL
LIN {X 0,Y 587.363,Z 358.314,A -85,B 0,C 180,E1 -1585.78,E2 -1585.78} C_VEL
LIN {X 0,Y 587.345,Z 358.32,A -85,B 0,C 180,E1 -1588.231,E2 -1588.231} C_VEL
LIN {X 0,Y 587.354,Z 358.323,A -85,B 0,C 180,E1 -1590.867,E2 -1590.867} C_VEL
LIN {X 0,Y 587.345,Z 358.317,A -85,B 0,C 180,E1 -1593.823,E2 -1593.823} C_VEL
LIN {X 0,Y 587.338,Z 358.32,A -85,B 0,C 180,E1 -1595.994,E2 -1595.994} C_VEL
LIN {X 0,Y 587.328,Z 358.324,A -85,B 0,C 180,E1 -1598.226,E2 -1598.226} C_VEL
LIN {X 0,Y 587.351,Z 358.317,A -85,B 0,C 180,E1 -1601.151,E2 -1601.151} C_VEL
LIN {X 0,Y 587.326,Z 358.324,A -85,B 0,C 180,E1 -1604.025,E2 -1604.025} C_VEL
LIN {X 0,Y 587.36,Z 358.321,A -85,B 0,C 180,E1 -1606.154,E2 -1606.154} C_VEL
LIN {X 0,Y 587.344,Z 358.318,A -85,B 0,C 180,E1 -1608.963,E2 -1608.963} C_VEL
LIN {X 0,Y 587.37,Z 358.317,A -85,B 0,C 180,E1 -1611.745,E2 -1611.745} C_VEL
LIN {X 0,Y 587.36,Z 358.32,A -85,B 0,C 180,E1 -1614.507,E2 -1614.507} C_VEL
LIN {X 0,Y 587.378,Z 358.312,A -85,B 0,C 180,E1 -1617.257,E2 -1617.257} C_VEL
LIN {X 0,Y 587.388,Z 358.321,A -85,B 0,C 180,E1 -1620,E2 -1620} C_VEL
LIN {X 0,Y 587.378,Z 358.314,A -85,B 0,C 180,E1 -1622.743,E2 -1622.743} C_VEL
LIN {X 0,Y 587.361,Z 358.318,A -85,B 0,C 180,E1 -1625.493,E2 -1625.493} C_VEL
LIN {X 0,Y 587.371,Z 358.318,A -85,B 0,C 180,E1 -1628.255,E2 -1628.255} C_VEL
LIN {X 0,Y 587.354,Z 358.317,A -85,B 0,C 180,E1 -1631.134,E2 -1631.134} C_VEL
LIN {X 0,Y 587.371,Z 358.317,A -85,B 0,C 180,E1 -1634.26,E2 -1634.26} C_VEL
LIN {X 0,Y 587.354,Z 358.321,A -85,B 0,C 180,E1 -1637.406,E2 -1637.406} C_VEL
LIN {X 0,Y 587.313,Z 358.323,A -85,B 0,C 180,E1 -1638.311,E2 -1638.311} C_VEL
LIN {X 0,Y 586.671,Z 358.402,A -85,B 0,C 180,E1 -1638.884,E2 -1638.884} C_VEL
LIN {X 0,Y 583.847,Z 358.761,A -85,B 0,C 180,E1 -1639.812,E2 -1639.812} C_VEL
LIN {X 0,Y 581.437,Z 359.063,A -85,B 0,C 180,E1 -1640.559,E2 -1640.559} C_VEL
LIN {X 0,Y 580.384,Z 359.191,A -85,B 0,C 180,E1 -1641.136,E2 -1641.136} C_VEL
LIN {X 0,Y 580.289,Z 359.201,A -85,B 0,C 180,E1 -1641.331,E2 -1641.331} C_VEL
LIN {X 0,Y 580.306,Z 359.195,A -85,B 0,C 180,E1 -1644.316,E2 -1644.316} C_VEL
LIN {X 0,Y 580.282,Z 359.198,A -85,B 0,C 180,E1 -1646.623,E2 -1646.623} C_VEL
LIN {X 0,Y 580.307,Z 359.202,A -85,B 0,C 180,E1 -1649.31,E2 -1649.31} C_VEL
LIN {X 0,Y 580.333,Z 359.203,A -85,B 0,C 180,E1 -1652.353,E2 -1652.353} C_VEL
LIN {X 0,Y 580.49,Z 367.697,A -85,B 0,C 180,E1 -1653.843,E2 -1653.843} C_VEL
LIN {X 0,Y 580.403,Z 384.056,A -85,B 0,C 180,E1 -1656.668,E2 -1656.668} C_VEL
LIN {X 0,Y 580.312,Z 394.167,A -85,B 0,C 180,E1 -1658.393,E2 -1658.393} C_VEL
LIN {X 0,Y 580.979,Z 399.44,A -85,B 0,C 180,E1 -1658.479,E2 -1658.479} C_VEL
LIN {X 0,Y 580.816,Z 501.02,A -85,B 0,C 180,E1 -1659.755,E2 -1659.755} C_VEL
LIN {X 0,Y 580.722,Z 514.38,A -85,B 0,C 180,E1 -1660.065,E2 -1660.065} C_VEL
LIN {X 0,Y 580.646,Z 526.937,A -85,B 0,C 180,E1 -1660.503,E2 -1660.503} C_VEL
LIN {X 0,Y 580.555,Z 538.082,A -85,B 0,C 180,E1 -1661.025,E2 -1661.025} C_VEL
LIN {X 0,Y 580.468,Z 548.261,A -85,B 0,C 180,E1 -1661.626,E2 -1661.626} C_VEL
LIN {X 0,Y 580.359,Z 558.572,A -85,B 0,C 180,E1 -1662.379,E2 -1662.379} C_VEL
LIN {X 0,Y 580.268,Z 569.076,A -85,B 0,C 180,E1 -1663.334,E2 -1663.334} C_VEL
LIN {X 0,Y 580.228,Z 576.853,A -85,B 0,C 180,E1 -1664.202,E2 -1664.202} C_VEL
LIN {X 0,Y 580.156,Z 584.103,A -85,B 0,C 180,E1 -1665.181,E2 -1665.181} C_VEL
LIN {X 0,Y 580.118,Z 590.873,A -85,B 0,C 180,E1 -1666.326,E2 -1666.326} C_VEL
LIN {X 0,Y 580.089,Z 595.347,A -85,B 0,C 180,E1 -1667.276,E2 -1667.276} C_VEL
LIN {X 0,Y 580.094,Z 598.864,A -85,B 0,C 180,E1 -1668.214,E2 -1668.214} C_VEL
LIN {X 0,Y 580.031,Z 601.472,A -85,B 0,C 180,E1 -1669.133,E2 -1669.133} C_VEL
LIN {X 0,Y 580.046,Z 603.335,A -85,B 0,C 180,E1 -1670.046,E2 -1670.046} C_VEL
LIN {X 0,Y 580.011,Z 604.501,A -85,B 0,C 180,E1 -1670.943,E2 -1670.943} C_VEL
LIN {X 0,Y 580.021,Z 604.987,A -85,B 0,C 180,E1 -1671.962,E2 -1671.962} C_VEL
LIN {X 0,Y 580.036,Z 604.54,A -85,B 0,C 180,E1 -1673.101,E2 -1673.101} C_VEL
LIN {X 0,Y 580.049,Z 602.618,A -85,B 0,C 180,E1 -1674.438,E2 -1674.438} C_VEL
LIN {X 0,Y 580.075,Z 600.09,A -85,B 0,C 180,E1 -1675.474,E2 -1675.474} C_VEL
LIN {X 0,Y 580.089,Z 595.746,A -85,B 0,C 180,E1 -1676.717,E2 -1676.717} C_VEL
LIN {X 0,Y 580.148,Z 590.738,A -85,B 0,C 180,E1 -1677.789,E2 -1677.789} C_VEL
LIN {X 0,Y 580.186,Z 583.517,A -85,B 0,C 180,E1 -1678.995,E2 -1678.995} C_VEL
LIN {X 0,Y 580.232,Z 575.734,A -85,B 0,C 180,E1 -1680.023,E2 -1680.023} C_VEL
LIN {X 0,Y 580.31,Z 566.368,A -85,B 0,C 180,E1 -1681.024,E2 -1681.024} C_VEL
LIN {X 0,Y 580.396,Z 556.033,A -85,B 0,C 180,E1 -1681.911,E2 -1681.911} C_VEL
LIN {X 0,Y 580.522,Z 544.404,A -85,B 0,C 180,E1 -1682.707,E2 -1682.707} C_VEL
LIN {X 0,Y 580.6,Z 532.5,A -85,B 0,C 180,E1 -1683.343,E2 -1683.343} C_VEL
LIN {X 0,Y 580.672,Z 520.231,A -85,B 0,C 180,E1 -1683.839,E2 -1683.839} C_VEL
LIN {X 0,Y 580.764,Z 506.748,A -85,B 0,C 180,E1 -1684.221,E2 -1684.221} C_VEL
LIN {X 0,Y 580.815,Z 492.977,A -85,B 0,C 180,E1 -1684.452,E2 -1684.452} C_VEL
LIN {X 0,Y 580.816,Z 397.158,A -85,B 0,C 180,E1 -1685.643,E2 -1685.643} C_VEL
LIN {X 0,Y 580.323,Z 394.1,A -85,B 0,C 180,E1 -1685.708,E2 -1685.708} C_VEL
LIN {X 0,Y 580.457,Z 376.62,A -85,B 0,C 180,E1 -1688.7,E2 -1688.7} C_VEL
LIN {X 0,Y 580.534,Z 360.685,A -85,B 0,C 180,E1 -1691.47,E2 -1691.47} C_VEL
LIN {X 0,Y 580.311,Z 359.199,A -85,B 0,C 180,E1 -1691.783,E2 -1691.783} C_VEL
LIN {X 0,Y 580.3,Z 359.204,A -85,B 0,C 180,E1 -1694.547,E2 -1694.547} C_VEL
LIN {X 0,Y 580.281,Z 359.206,A -85,B 0,C 180,E1 -1696.695,E2 -1696.695} C_VEL
LIN {X 0,Y 580.305,Z 359.194,A -85,B 0,C 180,E1 -1699.533,E2 -1699.533} C_VEL
LIN {X 0,Y 580.335,Z 359.198,A -85,B 0,C 180,E1 -1702.344,E2 -1702.344} C_VEL
LIN {X 0,Y 580.333,Z 359.191,A -85,B 0,C 180,E1 -1705.136,E2 -1705.136} C_VEL
LIN {X 0,Y 580.346,Z 359.192,A -85,B 0,C 180,E1 -1707.917,E2 -1707.917} C_VEL
LIN {X 0,Y 580.366,Z 359.19,A -85,B 0,C 180,E1 -1710.693,E2 -1710.693} C_VEL
LIN {X 0,Y 580.283,Z 359.197,A -85,B 0,C 180,E1 -1713.471,E2 -1713.471} C_VEL
LIN {X 0,Y 580.324,Z 359.193,A -85,B 0,C 180,E1 -1715.559,E2 -1715.559} C_VEL
LIN {X 0,Y 580.329,Z 359.198,A -85,B 0,C 180,E1 -1718.355,E2 -1718.355} C_VEL
LIN {X 0,Y 580.303,Z 359.194,A -85,B 0,C 180,E1 -1721.19,E2 -1721.19} C_VEL
LIN {X 0,Y 580.328,Z 359.201,A -85,B 0,C 180,E1 -1724.016,E2 -1724.016} C_VEL
LIN {X 0,Y 580.314,Z 359.193,A -85,B 0,C 180,E1 -1726.913,E2 -1726.913} C_VEL
LIN {X 0,Y 580.288,Z 359.204,A -85,B 0,C 180,E1 -1729.822,E2 -1729.822} C_VEL
LIN {X 0,Y 580.27,Z 359.206,A -85,B 0,C 180,E1 -1732.052,E2 -1732.052} C_VEL
LIN {X 0,Y 580.307,Z 359.194,A -85,B 0,C 180,E1 -1735.079,E2 -1735.079} C_VEL
LIN {X 0,Y 580.3,Z 359.198,A -85,B 0,C 180,E1 -1738.184,E2 -1738.184} C_VEL
LIN {X 0,Y 580.297,Z 359.195,A -85,B 0,C 180,E1 -1740.696,E2 -1740.696} C_VEL
LIN {X 0,Y 580.301,Z 359.198,A -85,B 0,C 180,E1 -1743.315,E2 -1743.315} C_VEL
LIN {X 0,Y 580.325,Z 359.2,A -85,B 0,C 180,E1 -1745.767,E2 -1745.767} C_VEL
LIN {X 0,Y 580.285,Z 359.198,A -85,B 0,C 180,E1 -1748.145,E2 -1748.145} C_VEL
LIN {X 0,Y 580.297,Z 359.196,A -85,B 0,C 180,E1 -1750.842,E2 -1750.842} C_VEL
LIN {X 0,Y 580.283,Z 359.205,A -85,B 0,C 180,E1 -1753.656,E2 -1753.656} C_VEL
LIN {X 0,Y 580.287,Z 359.197,A -85,B 0,C 180,E1 -1756.606,E2 -1756.606} C_VEL
LIN {X 0,Y 580.348,Z 359.351,A -85,B 0,C 180,E1 -1758.379,E2 -1758.379} C_VEL
LIN {X 0,Y 580.517,Z 365.564,A -85,B 0,C 180,E1 -1759.473,E2 -1759.473} C_VEL
LIN {X 0,Y 580.384,Z 382.04,A -85,B 0,C 180,E1 -1762.321,E2 -1762.321} C_VEL
LIN {X 0,Y 580.315,Z 394.212,A -85,B 0,C 180,E1 -1764.398,E2 -1764.398} C_VEL
LIN {X 0,Y 580.95,Z 399.886,A -85,B 0,C 180,E1 -1764.484,E2 -1764.484} C_VEL
LIN {X 0,Y 580.786,Z 501.041,A -85,B 0,C 180,E1 -1765.758,E2 -1765.758} C_VEL
LIN {X 0,Y 580.732,Z 514.028,A -85,B 0,C 180,E1 -1766.055,E2 -1766.055} C_VEL
LIN {X 0,Y 580.67,Z 526.048,A -85,B 0,C 180,E1 -1766.468,E2 -1766.468} C_VEL
LIN {X 0,Y 580.571,Z 537.437,A -85,B 0,C 180,E1 -1766.993,E2 -1766.993} C_VEL
LIN {X 0,Y 580.477,Z 547.887,A -85,B 0,C 180,E1 -1767.605,E2 -1767.605} C_VEL
LIN {X 0,Y 580.39,Z 557.744,A -85,B 0,C 180,E1 -1768.316,E2 -1768.316} C_VEL
LIN {X 0,Y 580.294,Z 567.689,A -85,B 0,C 180,E1 -1769.196,E2 -1769.196} C_VEL
LIN {X 0,Y 580.201,Z 577.008,A -85,B 0,C 180,E1 -1770.222,E2 -1770.222} C_VEL
LIN {X 0,Y 580.172,Z 584.287,A -85,B 0,C 180,E1 -1771.215,E2 -1771.215} C_VEL
LIN {X 0,Y 580.101,Z 591.148,A -85,B 0,C 180,E1 -1772.381,E2 -1772.381} C_VEL
LIN {X 0,Y 580.128,Z 597.021,A -85,B 0,C 180,E1 -1773.696,E2 -1773.696} C_VEL
LIN {X 0,Y 580.048,Z 600.874,A -85,B 0,C 180,E1 -1774.908,E2 -1774.908} C_VEL
LIN {X 0,Y 580.023,Z 602.667,A -85,B 0,C 180,E1 -1775.671,E2 -1775.671} C_VEL
LIN {X 0,Y 580.025,Z 603.93,A -85,B 0,C 180,E1 -1776.431,E2 -1776.431} C_VEL
LIN {X 0,Y 580.062,Z 604.672,A -85,B 0,C 180,E1 -1777.188,E2 -1777.188} C_VEL
LIN {X 0,Y 580.031,Z 604.967,A -85,B 0,C 180,E1 -1777.938,E2 -1777.938} C_VEL
LIN {X 0,Y 580.055,Z 604.678,A -85,B 0,C 180,E1 -1778.894,E2 -1778.894} C_VEL
LIN {X 0,Y 580.047,Z 603.11,A -85,B 0,C 180,E1 -1780.168,E2 -1780.168} C_VEL
LIN {X 0,Y 580.055,Z 601.555,A -85,B 0,C 180,E1 -1780.914,E2 -1780.914} C_VEL
LIN {X 0,Y 580.081,Z 598.396,A -85,B 0,C 180,E1 -1782.004,E2 -1782.004} C_VEL
LIN {X 0,Y 580.117,Z 593.883,A -85,B 0,C 180,E1 -1783.146,E2 -1783.146} C_VEL
LIN {X 0,Y 580.127,Z 587.539,A -85,B 0,C 180,E1 -1784.362,E2 -1784.362} C_VEL
LIN {X 0,Y 580.196,Z 580.663,A -85,B 0,C 180,E1 -1785.398,E2 -1785.398} C_VEL
LIN {X 0,Y 580.237,Z 572.97,A -85,B 0,C 180,E1 -1786.338,E2 -1786.338} C_VEL
LIN {X 0,Y 580.342,Z 564.091,A -85,B 0,C 180,E1 -1787.232,E2 -1787.232} C_VEL
LIN {X 0,Y 580.41,Z 554.41,A -85,B 0,C 180,E1 -1788.032,E2 -1788.032} C_VEL
LIN {X 0,Y 580.506,Z 542.297,A -85,B 0,C 180,E1 -1788.831,E2 -1788.831} C_VEL
LIN {X 0,Y 580.621,Z 532.013,A -85,B 0,C 180,E1 -1789.363,E2 -1789.363} C_VEL
LIN {X 0,Y 580.672,Z 521.134,A -85,B 0,C 180,E1 -1789.804,E2 -1789.804} C_VEL
LIN {X 0,Y 580.748,Z 509.32,A -85,B 0,C 180,E1 -1790.158,E2 -1790.158} C_VEL
LIN {X 0,Y 580.806,Z 496.802,A -85,B 0,C 180,E1 -1790.4,E2 -1790.4} C_VEL
LIN {X 0,Y 580.83,Z 397.347,A -85,B 0,C 180,E1 -1791.64,E2 -1791.64} C_VEL
LIN {X 0,Y 580.33,Z 394.089,A -85,B 0,C 180,E1 -1791.71,E2 -1791.71} C_VEL
LIN {X 0,Y 580.442,Z 377.115,A -85,B 0,C 180,E1 -1794.616,E2 -1794.616} C_VEL
LIN {X 0,Y 580.559,Z 362.083,A -85,B 0,C 180,E1 -1797.224,E2 -1797.224} C_VEL
LIN {X 0,Y 580.307,Z 359.199,A -85,B 0,C 180,E1 -1797.744,E2 -1797.744} C_VEL
LIN {X 0,Y 580.342,Z 359.193,A -85,B 0,C 180,E1 -1800,E2 -1800} C_VEL
LIN {X 0,Y 580.34,Z 359.197,A -85,B 0,C 180,E1 -1802.776,E2 -1802.776} C_VEL
LIN {X 0,Y 580.318,Z 359.193,A -85,B 0,C 180,E1 -1805.56,E2 -1805.56} C_VEL
LIN {X 0,Y 580.327,Z 359.201,A -85,B 0,C 180,E1 -1808.356,E2 -1808.356} C_VEL
LIN {X 0,Y 580.322,Z 359.193,A -85,B 0,C 180,E1 -1811.208,E2 -1811.208} C_VEL
LIN {X 0,Y 580.317,Z 359.2,A -85,B 0,C 180,E1 -1814.017,E2 -1814.017} C_VEL
LIN {X 0,Y 580.307,Z 359.195,A -85,B 0,C 180,E1 -1816.916,E2 -1816.916} C_VEL
LIN {X 0,Y 580.301,Z 359.202,A -85,B 0,C 180,E1 -1819.822,E2 -1819.822} C_VEL
LIN {X 0,Y 580.321,Z 359.192,A -85,B 0,C 180,E1 -1822.801,E2 -1822.801} C_VEL
LIN {X 0,Y 580.303,Z 359.195,A -85,B 0,C 180,E1 -1825.08,E2 -1825.08} C_VEL
LIN {X 0,Y 580.312,Z 359.202,A -85,B 0,C 180,E1 -1827.864,E2 -1827.864} C_VEL
LIN {X 0,Y 580.292,Z 359.196,A -85,B 0,C 180,E1 -1830.698,E2 -1830.698} C_VEL
LIN {X 0,Y 580.3,Z 359.201,A -85,B 0,C 180,E1 -1833.318,E2 -1833.318} C_VEL
LIN {X 0,Y 580.318,Z 359.199,A -85,B 0,C 180,E1 -1835.768,E2 -1835.768} C_VEL
LIN {X 0,Y 580.282,Z 359.198,A -85,B 0,C 180,E1 -1838.147,E2 -1838.147} C_VEL
LIN {X 0,Y 580.295,Z 359.198,A -85,B 0,C 180,E1 -1840.844,E2 -1840.844} C_VEL
LIN {X 0,Y 580.284,Z 359.201,A -85,B 0,C 180,E1 -1843.658,E2 -1843.658} C_VEL
LIN {X 0,Y 580.271,Z 359.2,A -85,B 0,C 180,E1 -1846.61,E2 -1846.61} C_VEL
LIN {X 0,Y 580.295,Z 359.205,A -85,B 0,C 180,E1 -1849.158,E2 -1849.158} C_VEL
LIN {X 0,Y 580.287,Z 359.197,A -85,B 0,C 180,E1 -1851.928,E2 -1851.928} C_VEL
LIN {X 0,Y 580.306,Z 359.197,A -85,B 0,C 180,E1 -1854.458,E2 -1854.458} C_VEL
LIN {X 0,Y 580.288,Z 359.205,A -85,B 0,C 180,E1 -1856.976,E2 -1856.976} C_VEL
LIN {X 0,Y 580.308,Z 359.196,A -85,B 0,C 180,E1 -1859.427,E2 -1859.427} C_VEL
LIN {X 0,Y 580.318,Z 359.195,A -85,B 0,C 180,E1 -1862.138,E2 -1862.138} C_VEL
LIN {X 0,Y 580.308,Z 359.201,A -85,B 0,C 180,E1 -1864.922,E2 -1864.922} C_VEL
LIN {X 0,Y 580.317,Z 359.366,A -85,B 0,C 180,E1 -1867.106,E2 -1867.106} C_VEL
LIN {X 0,Y 580.918,Z 363.769,A -85,B 0,C 180,E1 -1867.787,E2 -1867.787} C_VEL
LIN {X 0,Y 580.7,Z 383.859,A -85,B 0,C 180,E1 -1870.736,E2 -1870.736} C_VEL
LIN {X 0,Y 580.543,Z 402.808,A -85,B 0,C 180,E1 -1873.473,E2 -1873.473} C_VEL
LIN {X 0,Y 580.372,Z 422.8,A -85,B 0,C 180,E1 -1876.32,E2 -1876.32} C_VEL
LIN {X 0,Y 580.987,Z 426.803,A -85,B 0,C 180,E1 -1876.402,E2 -1876.402} C_VEL
LIN {X 0,Y 580.831,Z 530.999,A -85,B 0,C 180,E1 -1877.71,E2 -1877.71} C_VEL
LIN {X 0,Y 580.725,Z 544.255,A -85,B 0,C 180,E1 -1878.018,E2 -1878.018} C_VEL
LIN {X 0,Y 580.624,Z 557.15,A -85,B 0,C 180,E1 -1878.466,E2 -1878.466} C_VEL
LIN {X 0,Y 580.567,Z 568.648,A -85,B 0,C 180,E1 -1879.01,E2 -1879.01} C_VEL
LIN {X 0,Y 580.444,Z 580.218,A -85,B 0,C 180,E1 -1879.713,E2 -1879.713} C_VEL
LIN {X 0,Y 580.341,Z 590.611,A -85,B 0,C 180,E1 -1880.504,E2 -1880.504} C_VEL
LIN {X 0,Y 580.271,Z 599.122,A -85,B 0,C 180,E1 -1881.293,E2 -1881.293} C_VEL
LIN {X 0,Y 580.221,Z 606.969,A -85,B 0,C 180,E1 -1882.169,E2 -1882.169} C_VEL
LIN {X 0,Y 580.153,Z 614.655,A -85,B 0,C 180,E1 -1883.222,E2 -1883.222} C_VEL
LIN {X 0,Y 580.139,Z 621.685,A -85,B 0,C 180,E1 -1884.439,E2 -1884.439} C_VEL
LIN {X 0,Y 580.108,Z 626.376,A -85,B 0,C 180,E1 -1885.484,E2 -1885.484} C_VEL
LIN {X 0,Y 580.123,Z 629.96,A -85,B 0,C 180,E1 -1886.528,E2 -1886.528} C_VEL
LIN {X 0,Y 580.043,Z 631.811,A -85,B 0,C 180,E1 -1887.223,E2 -1887.223} C_VEL
LIN {X 0,Y 580.038,Z 633.201,A -85,B 0,C 180,E1 -1887.918,E2 -1887.918} C_VEL
LIN {X 0,Y 580.04,Z 634.785,A -85,B 0,C 180,E1 -1889.307,E2 -1889.307} C_VEL
LIN {X 0,Y 580.037,Z 635,A -85,B 0,C 180,E1 -1890.001,E2 -1890.001} C_VEL
LIN {X 0,Y 580.047,Z 634.185,A -85,B 0,C 180,E1 -1891.389,E2 -1891.389} C_VEL
LIN {X 0,Y 580.039,Z 633.199,A -85,B 0,C 180,E1 -1892.084,E2 -1892.084} C_VEL
LIN {X 0,Y 580.043,Z 631.808,A -85,B 0,C 180,E1 -1892.779,E2 -1892.779} C_VEL
LIN {X 0,Y 580.109,Z 628.893,A -85,B 0,C 180,E1 -1893.821,E2 -1893.821} C_VEL
LIN {X 0,Y 580.054,Z 624.946,A -85,B 0,C 180,E1 -1894.866,E2 -1894.866} C_VEL
LIN {X 0,Y 580.139,Z 618.872,A -85,B 0,C 180,E1 -1896.086,E2 -1896.086} C_VEL
LIN {X 0,Y 580.185,Z 612.231,A -85,B 0,C 180,E1 -1897.133,E2 -1897.133} C_VEL
LIN {X 0,Y 580.251,Z 603.983,A -85,B 0,C 180,E1 -1898.183,E2 -1898.183} C_VEL
LIN {X 0,Y 580.308,Z 595.529,A -85,B 0,C 180,E1 -1899.059,E2 -1899.059} C_VEL
LIN {X 0,Y 580.417,Z 585.086,A -85,B 0,C 180,E1 -1899.937,E2 -1899.937} C_VEL
LIN {X 0,Y 580.507,Z 574.743,A -85,B 0,C 180,E1 -1900.64,E2 -1900.64} C_VEL
LIN {X 0,Y 580.598,Z 563.225,A -85,B 0,C 180,E1 -1901.265,E2 -1901.265} C_VEL
LIN {X 0,Y 580.666,Z 550.448,A -85,B 0,C 180,E1 -1901.786,E2 -1901.786} C_VEL
LIN {X 0,Y 580.768,Z 537.401,A -85,B 0,C 180,E1 -1902.16,E2 -1902.16} C_VEL
LIN {X 0,Y 580.845,Z 525.024,A -85,B 0,C 180,E1 -1902.381,E2 -1902.381} C_VEL
LIN {X 0,Y 580.876,Z 425.985,A -85,B 0,C 180,E1 -1903.611,E2 -1903.611} C_VEL
LIN {X 0,Y 580.374,Z 422.787,A -85,B 0,C 180,E1 -1903.682,E2 -1903.682} C_VEL
LIN {X 0,Y 580.525,Z 402.795,A -85,B 0,C 180,E1 -1906.53,E2 -1906.53} C_VEL
LIN {X 0,Y 580.702,Z 383.854,A -85,B 0,C 180,E1 -1909.265,E2 -1909.265} C_VEL
LIN {X 0,Y 580.885,Z 365.015,A -85,B 0,C 180,E1 -1912.029,E2 -1912.029} C_VEL
LIN {X 0,Y 580.458,Z 359.978,A -85,B 0,C 180,E1 -1912.796,E2 -1912.796} C_VEL
LIN {X 0,Y 580.29,Z 359.205,A -85,B 0,C 180,E1 -1912.927,E2 -1912.927} C_VEL
LIN {X 0,Y 580.313,Z 359.2,A -85,B 0,C 180,E1 -1915.08,E2 -1915.08} C_VEL
LIN {X 0,Y 580.303,Z 359.196,A -85,B 0,C 180,E1 -1918.186,E2 -1918.186} C_VEL
LIN {X 0,Y 580.298,Z 359.198,A -85,B 0,C 180,E1 -1920.696,E2 -1920.696} C_VEL
LIN {X 0,Y 580.309,Z 359.203,A -85,B 0,C 180,E1 -1923.317,E2 -1923.317} C_VEL
LIN {X 0,Y 580.255,Z 359.203,A -85,B 0,C 180,E1 -1925.757,E2 -1925.757} C_VEL
LIN {X 0,Y 580.294,Z 359.196,A -85,B 0,C 180,E1 -1928.147,E2 -1928.147} C_VEL
LIN {X 0,Y 580.303,Z 359.201,A -85,B 0,C 180,E1 -1930.844,E2 -1930.844} C_VEL
LIN {X 0,Y 580.284,Z 359.199,A -85,B 0,C 180,E1 -1933.658,E2 -1933.658} C_VEL
LIN {X 0,Y 580.283,Z 359.202,A -85,B 0,C 180,E1 -1936.61,E2 -1936.61} C_VEL
LIN {X 0,Y 580.302,Z 359.2,A -85,B 0,C 180,E1 -1939.157,E2 -1939.157} C_VEL
LIN {X 0,Y 580.293,Z 359.196,A -85,B 0,C 180,E1 -1941.928,E2 -1941.928} C_VEL
LIN {X 0,Y 580.254,Z 359.205,A -85,B 0,C 180,E1 -1944.453,E2 -1944.453} C_VEL
LIN {X 0,Y 580.295,Z 359.202,A -85,B 0,C 180,E1 -1946.975,E2 -1946.975} C_VEL
LIN {X 0,Y 580.299,Z 359.195,A -85,B 0,C 180,E1 -1949.425,E2 -1949.425} C_VEL
LIN {X 0,Y 580.296,Z 359.198,A -85,B 0,C 180,E1 -1952.143,E2 -1952.143} C_VEL
LIN {X 0,Y 580.31,Z 359.198,A -85,B 0,C 180,E1 -1954.92,E2 -1954.92} C_VEL
LIN {X 0,Y 580.278,Z 359.198,A -85,B 0,C 180,E1 -1957.948,E2 -1957.948} C_VEL
LIN {X 0,Y 580.305,Z 359.196,A -85,B 0,C 180,E1 -1960.914,E2 -1960.914} C_VEL
LIN {X 0,Y 580.281,Z 359.199,A -85,B 0,C 180,E1 -1963.826,E2 -1963.826} C_VEL
LIN {X 0,Y 580.329,Z 359.194,A -85,B 0,C 180,E1 -1965.983,E2 -1965.983} C_VEL
LIN {X 0,Y 580.311,Z 359.195,A -85,B 0,C 180,E1 -1968.827,E2 -1968.827} C_VEL
LIN {X 0,Y 580.332,Z 359.192,A -85,B 0,C 180,E1 -1971.644,E2 -1971.644} C_VEL
LIN {X 0,Y 580.327,Z 359.197,A -85,B 0,C 180,E1 -1974.44,E2 -1974.44} C_VEL
LIN {X 0,Y 580.344,Z 359.188,A -85,B 0,C 180,E1 -1977.224,E2 -1977.224} C_VEL
LIN {X 0,Y 580.358,Z 359.197,A -85,B 0,C 180,E1 -1980,E2 -1980} C_VEL
LIN {X 0,Y 580.344,Z 359.19,A -85,B 0,C 180,E1 -1982.777,E2 -1982.777} C_VEL
LIN {X 0,Y 580.328,Z 359.195,A -85,B 0,C 180,E1 -1985.56,E2 -1985.56} C_VEL
LIN {X 0,Y 580.333,Z 359.194,A -85,B 0,C 180,E1 -1988.356,E2 -1988.356} C_VEL
LIN {X 0,Y 580.306,Z 359.196,A -85,B 0,C 180,E1 -1991.191,E2 -1991.191} C_VEL
LIN {X 0,Y 580.331,Z 359.197,A -85,B 0,C 180,E1 -1994.017,E2 -1994.017} C_VEL
LIN {X 0,Y 580.318,Z 359.193,A -85,B 0,C 180,E1 -1996.914,E2 -1996.914} C_VEL
LIN {X 0,Y 580.309,Z 359.201,A -85,B 0,C 180,E1 -1999.822,E2 -1999.822} C_VEL
LIN {X 0,Y 580.289,Z 359.201,A -85,B 0,C 180,E1 -2001.331,E2 -2001.331} C_VEL
LIN {X 0,Y 579.592,Z 359.289,A -85,B 0,C 180,E1 -2001.91,E2 -2001.91} C_VEL
LIN {X 0,Y 576.715,Z 359.643,A -85,B 0,C 180,E1 -2002.85,E2 -2002.85} C_VEL
LIN {X 0,Y 574.32,Z 359.949,A -85,B 0,C 180,E1 -2003.606,E2 -2003.606} C_VEL
LIN {X 0,Y 573.322,Z 360.067,A -85,B 0,C 180,E1 -2004.19,E2 -2004.19} C_VEL
LIN {X 0,Y 573.255,Z 360.073,A -85,B 0,C 180,E1 -2004.387,E2 -2004.387} C_VEL
LIN {X 0,Y 573.254,Z 360.076,A -85,B 0,C 180,E1 -2006.976,E2 -2006.976} C_VEL
LIN {X 0,Y 573.253,Z 360.083,A -85,B 0,C 180,E1 -2009.488,E2 -2009.488} C_VEL
LIN {X 0,Y 573.298,Z 360.225,A -85,B 0,C 180,E1 -2012.283,E2 -2012.283} C_VEL
LIN {X 0,Y 573.513,Z 365.67,A -85,B 0,C 180,E1 -2013.256,E2 -2013.256} C_VEL
LIN {X 0,Y 573.377,Z 381.559,A -85,B 0,C 180,E1 -2016.04,E2 -2016.04} C_VEL
LIN {X 0,Y 573.289,Z 394.294,A -85,B 0,C 180,E1 -2018.229,E2 -2018.229} C_VEL
